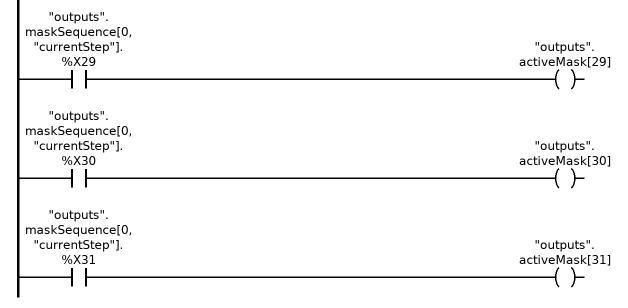
   RUNG wire#powerrail
      Contact( "outputs".maskSequence[0, "currentStep"].%X0 )
      Coil( "outputs".activeMask[0] )
   END_RUNG
   RUNG wire#powerrail
      Contact( "outputs".maskSequence[0, "currentStep"].%X1 )
      Coil( "outputs".activeMask[1] )
   END_RUNG
   RUNG wire#powerrail
      Contact( "outputs".maskSequence[0, "currentStep"].%X2 )
      Coil( "outputs".activeMask[2] )
   END_RUNG
   RUNG wire#powerrail
      Contact( "outputs".maskSequence[0, "currentStep"].%X3 )
      Coil( "outputs".activeMask[3] )
   END_RUNG
   RUNG wire#powerrail
      Contact( "outputs".maskSequence[0, "currentStep"].%X4 )
      Coil( "outputs".activeMask[4] )
   END_RUNG
   RUNG wire#powerrail
      Contact( "outputs".maskSequence[0, "currentStep"].%X5 )
      Coil( "outputs".activeMask[5] )
   END_RUNG
   RUNG wire#powerrail
      Contact( "outputs".maskSequence[0, "currentStep"].%X6 )
      Coil( "outputs".activeMask[6] )
   END_RUNG
   RUNG wire#powerrail
      Contact( "outputs".maskSequence[0, "currentStep"].%X7 )
      Coil( "outputs".activeMask[7] )
   END_RUNG
   RUNG wire#powerrail
      Contact( "outputs".maskSequence[0, "currentStep"].%X8 )
      Coil( "outputs".activeMask[8] )
   END_RUNG
   RUNG wire#powerrail
      Contact( "outputs".maskSequence[0, "currentStep"].%X9 )
      Coil( "outputs".activeMask[9] )
   END_RUNG
   RUNG wire#powerrail
      Contact( "outputs".maskSequence[0, "currentStep"].%X10 )
      Coil( "outputs".activeMask[10] )
   END_RUNG
   RUNG wire#powerrail
      Contact( "outputs".maskSequence[0, "currentStep"].%X11 )
      Coil( "outputs".activeMask[11] )
   END_RUNG
   RUNG wire#powerrail
      Contact( "outputs".maskSequence[0, "currentStep"].%X12 )
      Coil( "outputs".activeMask[12] )
   END_RUNG
   RUNG wire#powerrail
      Contact( "outputs".maskSequence[0, "currentStep"].%X13 )
      Coil( "outputs".activeMask[13] )
   END_RUNG
   RUNG wire#powerrail
      Contact( "outputs".maskSequence[0, "currentStep"].%X14 )
      Coil( "outputs".activeMask[14] )
   END_RUNG
   RUNG wire#powerrail
      Contact( "outputs".maskSequence[0, "currentStep"].%X15 )
      Coil( "outputs".activeMask[15] )
   END_RUNG
   RUNG wire#powerrail
      Contact( "outputs".maskSequence[0, "currentStep"].%X16 )
      Coil( "outputs".activeMask[16] )
   END_RUNG
   RUNG wire#powerrail
      Contact( "outputs".maskSequence[0, "currentStep"].%X17 )
      Coil( "outputs".activeMask[17] )
   END_RUNG
   RUNG wire#powerrail
      Contact( "outputs".maskSequence[0, "currentStep"].%X18 )
      Coil( "outputs".activeMask[18] )
   END_RUNG
   RUNG wire#powerrail
      Contact( "outputs".maskSequence[0, "currentStep"].%X19 )
      Coil( "outputs".activeMask[19] )
   END_RUNG
   RUNG wire#powerrail
      Contact( "outputs".maskSequence[0, "currentStep"].%X20 )
      Coil( "outputs".activeMask[20] )
   END_RUNG
   RUNG wire#powerrail
      Contact( "outputs".maskSequence[0, "currentStep"].%X21 )
      Coil( "outputs".activeMask[21] )
   END_RUNG
   RUNG wire#powerrail
      Contact( "outputs".maskSequence[0, "currentStep"].%X22 )
      Coil( "outputs".activeMask[22] )
   END_RUNG
   RUNG wire#powerrail
      Contact( "outputs".maskSequence[0, "currentStep"].%X23 )
      Coil( "outputs".activeMask[23] )
   END_RUNG
   RUNG wire#powerrail
      Contact( "outputs".maskSequence[0, "currentStep"].%X24 )
      Coil( "outputs".activeMask[24] )
   END_RUNG
   RUNG wire#powerrail
      Contact( "outputs".maskSequence[0, "currentStep"].%X25 )
      Coil( "outputs".activeMask[25] )
   END_RUNG
   RUNG wire#powerrail
      Contact( "outputs".maskSequence[0, "currentStep"].%X26 )
      Coil( "outputs".activeMask[26] )
   END_RUNG
   RUNG wire#powerrail
      Contact( "outputs".maskSequence[0, "currentStep"].%X27 )
      Coil( "outputs".activeMask[27] )
   END_RUNG
   RUNG wire#powerrail
      Contact( "outputs".maskSequence[0, "currentStep"].%X28 )
      Coil( "outputs".activeMask[28] )
   END_RUNG
   RUNG wire#powerrail
      Contact( "outputs".maskSequence[0, "currentStep"].%X29 )
      Coil( "outputs".activeMask[29] )
   END_RUNG
   RUNG wire#powerrail
      Contact( "outputs".maskSequence[0, "currentStep"].%X30 )
      Coil( "outputs".activeMask[30] )
   END_RUNG
   RUNG wire#powerrail
      Contact( "outputs".maskSequence[0, "currentStep"].%X31 )
      Coil( "outputs".activeMask[31] )
   END_RUNG
   // the same network as SCL:
   "outputs".activeMask[0] := "outputs".maskSequence[0, "currentStep"].%X0;
   "outputs".activeMask[1] := "outputs".maskSequence[0, "currentStep"].%X1;
   "outputs".activeMask[2] := "outputs".maskSequence[0, "currentStep"].%X2;
   "outputs".activeMask[3] := "outputs".maskSequence[0, "currentStep"].%X3;
   "outputs".activeMask[4] := "outputs".maskSequence[0, "currentStep"].%X4;
   "outputs".activeMask[5] := "outputs".maskSequence[0, "currentStep"].%X5;
   "outputs".activeMask[6] := "outputs".maskSequence[0, "currentStep"].%X6;
   "outputs".activeMask[7] := "outputs".maskSequence[0, "currentStep"].%X7;
   "outputs".activeMask[8] := "outputs".maskSequence[0, "currentStep"].%X8;
   "outputs".activeMask[9] := "outputs".maskSequence[0, "currentStep"].%X9;
   "outputs".activeMask[10] := "outputs".maskSequence[0, "currentStep"].%X10;
   "outputs".activeMask[11] := "outputs".maskSequence[0, "currentStep"].%X11;
   "outputs".activeMask[12] := "outputs".maskSequence[0, "currentStep"].%X12;
   "outputs".activeMask[13] := "outputs".maskSequence[0, "currentStep"].%X13;
   "outputs".activeMask[14] := "outputs".maskSequence[0, "currentStep"].%X14;
   "outputs".activeMask[15] := "outputs".maskSequence[0, "currentStep"].%X15;
   "outputs".activeMask[16] := "outputs".maskSequence[0, "currentStep"].%X16;
   "outputs".activeMask[17] := "outputs".maskSequence[0, "currentStep"].%X17;
   "outputs".activeMask[18] := "outputs".maskSequence[0, "currentStep"].%X18;
   "outputs".activeMask[19] := "outputs".maskSequence[0, "currentStep"].%X19;
   "outputs".activeMask[20] := "outputs".maskSequence[0, "currentStep"].%X20;
   "outputs".activeMask[21] := "outputs".maskSequence[0, "currentStep"].%X21;
   "outputs".activeMask[22] := "outputs".maskSequence[0, "currentStep"].%X22;
   "outputs".activeMask[23] := "outputs".maskSequence[0, "currentStep"].%X23;
   "outputs".activeMask[24] := "outputs".maskSequence[0, "currentStep"].%X24;
   "outputs".activeMask[25] := "outputs".maskSequence[0, "currentStep"].%X25;
   "outputs".activeMask[26] := "outputs".maskSequence[0, "currentStep"].%X26;
   "outputs".activeMask[27] := "outputs".maskSequence[0, "currentStep"].%X27;
   "outputs".activeMask[28] := "outputs".maskSequence[0, "currentStep"].%X28;
   "outputs".activeMask[29] := "outputs".maskSequence[0, "currentStep"].%X29;
   "outputs".activeMask[30] := "outputs".maskSequence[0, "currentStep"].%X30;
   "outputs".activeMask[31] := "outputs".maskSequence[0, "currentStep"].%X31;
END_REGION
END_FUNCTION

FUNCTION "production" : Void   // FC15, LAD
{ S7_Optimized_Access := 'TRUE' }
VERSION : 0.1
// stored: AutoNumber true, IsIECCheckEnabled false, SetENOAutomatically false, UDAEnableTagReadback false
   VAR_TEMP   // added for the SCL form of the ladder/FBD networks
      _w1 : Bool;
      _w2 : Bool;
      _w3 : Bool;
   END_VAR
BEGIN

REGION Network 1: SHIFTS PRODUCTION
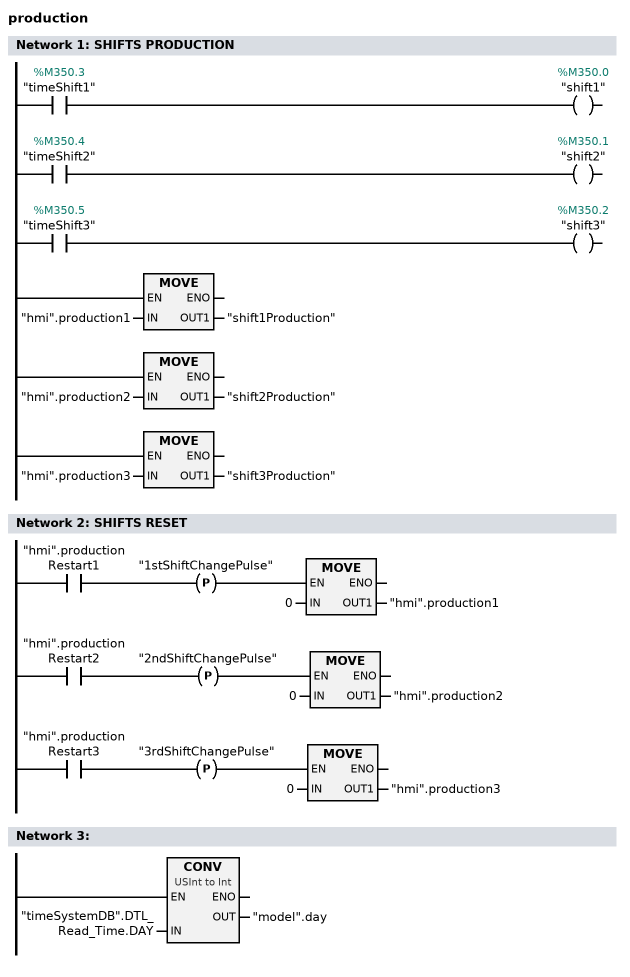
   RUNG wire#powerrail
      Contact( "timeShift1" )
      Coil( "shift1" )
   END_RUNG
   RUNG wire#powerrail
      Contact( "timeShift2" )
      Coil( "shift2" )
   END_RUNG
   RUNG wire#powerrail
      Contact( "timeShift3" )
      Coil( "shift3" )
   END_RUNG
   RUNG wire#powerrail
      Move(in := "hmi".production1, out1 => "shift1Production")
   END_RUNG
   RUNG wire#powerrail
      Move(in := "hmi".production2, out1 => "shift2Production")
   END_RUNG
   RUNG wire#powerrail
      Move(in := "hmi".production3, out1 => "shift3Production")
   END_RUNG
   // the same network as SCL:
   "shift1" := "timeShift1";
   "shift2" := "timeShift2";
   "shift3" := "timeShift3";
   "shift1Production" := "hmi".production1;
   "shift2Production" := "hmi".production2;
   "shift3Production" := "hmi".production3;
END_REGION

REGION Network 2: SHIFTS RESET
   RUNG wire#powerrail
      Contact( "hmi".productionRestart1 )
      P_Trig( "1stShiftChangePulse" )
      Move(in := 0, out1 => "hmi".production1)
   END_RUNG
   RUNG wire#powerrail
      Contact( "hmi".productionRestart2 )
      P_Trig( "2ndShiftChangePulse" )
      Move(in := 0, out1 => "hmi".production2)
   END_RUNG
   RUNG wire#powerrail
      Contact( "hmi".productionRestart3 )
      P_Trig( "3rdShiftChangePulse" )
      Move(in := 0, out1 => "hmi".production3)
   END_RUNG
   // the same network as SCL:
   #_w1 := "hmi".productionRestart1 AND NOT "1stShiftChangePulse";   // rising edge
   "1stShiftChangePulse" := "hmi".productionRestart1;
   IF #_w1 THEN "hmi".production1 := 0; END_IF;
   #_w2 := "hmi".productionRestart2 AND NOT "2ndShiftChangePulse";   // rising edge
   "2ndShiftChangePulse" := "hmi".productionRestart2;
   IF #_w2 THEN "hmi".production2 := 0; END_IF;
   #_w3 := "hmi".productionRestart3 AND NOT "3rdShiftChangePulse";   // rising edge
   "3rdShiftChangePulse" := "hmi".productionRestart3;
   IF #_w3 THEN "hmi".production3 := 0; END_IF;
END_REGION

REGION Network 3
   RUNG wire#powerrail
      { S7_Templates := "[SrcType := USInt, DestType := Int]" } Convert(in := "timeSystemDB".DTL_Read_Time.DAY, out => "model".day)
   END_RUNG
   // the same network as SCL:
   "model".day := USINT_TO_INT("timeSystemDB".DTL_Read_Time.DAY);
END_REGION
END_FUNCTION

FUNCTION "scannerConfiguration" : Void   // FC11, LAD
{ S7_Optimized_Access := 'TRUE' }
VERSION : 0.1
// stored: AutoNumber true, IsIECCheckEnabled false, SetENOAutomatically false, UDAEnableTagReadback false
   VAR_TEMP
      tempScannerOk1 : Bool;
      tempScannerOk2 : Bool;
      tempScannerOk3 : Bool;
   END_VAR
   VAR_TEMP   // added for the SCL form of the ladder/FBD networks
      _w1 : Bool;
      _w2 : Bool;
      _w3 : Bool;
      _w4 : Bool;
      _w5 : Bool;
      _w6 : Bool;
      _w7 : Bool;
      _w8 : Bool;
      _w9 : Bool;
      _w10 : Bool;
      _w11 : Bool;
      _w12 : Bool;
      _w13 : Bool;
      _w14 : Bool;
      _w15 : Bool;
   END_VAR
BEGIN

REGION Network 1: PORT CONFIGURATION
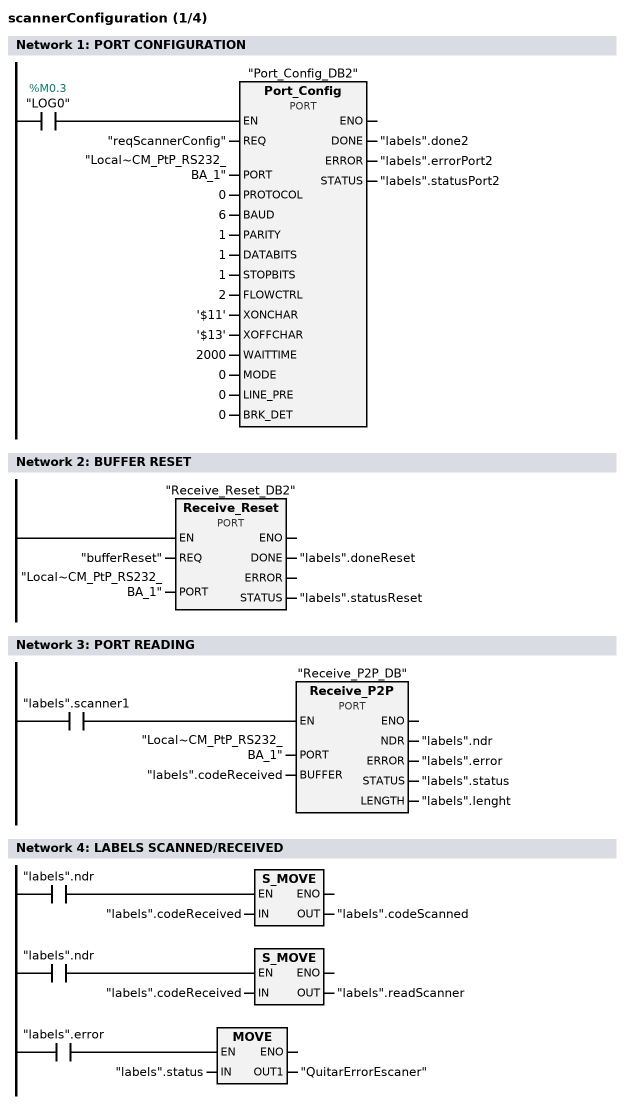
   RUNG wire#powerrail
      Contact( "LOG0" )
      { S7_Templates := "[card := 0, port_type := PORT, word_type := UInt, byte_type := USInt]" } "Port_Config_DB2".Port_Config(REQ := "reqScannerConfig", PORT := "Local~CM_PtP_RS232_BA_1", PROTOCOL := 0, BAUD := 6, PARITY := 1, DATABITS := 1, STOPBITS := 1, FLOWCTRL := 2, XONCHAR := '$11', XOFFCHAR := '$13', WAITTIME := 2000, MODE := 0, LINE_PRE := 0, BRK_DET := 0, DONE => "labels".done2, ERROR => "labels".errorPort2, STATUS => "labels".statusPort2)
   END_RUNG
   // the same network as SCL:
   IF "LOG0" THEN
       "Port_Config_DB2"(REQ := "reqScannerConfig",   // Port_Config
                         PORT := "Local~CM_PtP_RS232_BA_1",
                         PROTOCOL := 0,
                         BAUD := 6,
                         PARITY := 1,
                         DATABITS := 1,
                         STOPBITS := 1,
                         FLOWCTRL := 2,
                         XONCHAR := '$11',
                         XOFFCHAR := '$13',
                         WAITTIME := 2000,
                         MODE := 0,
                         LINE_PRE := 0,
                         BRK_DET := 0,
                         DONE => "labels".done2,
                         ERROR => "labels".errorPort2,
                         STATUS => "labels".statusPort2);
   END_IF;
END_REGION

REGION Network 2: BUFFER RESET
   RUNG wire#powerrail
      { S7_Templates := "[card := 0, port_type := PORT]" } "Receive_Reset_DB2".Receive_Reset(REQ := "bufferReset", PORT := "Local~CM_PtP_RS232_BA_1", DONE => "labels".doneReset, ERROR =>, STATUS => "labels".statusReset)
   END_RUNG
   // the same network as SCL:
   "Receive_Reset_DB2"(REQ := "bufferReset",   // Receive_Reset
                       PORT := "Local~CM_PtP_RS232_BA_1",
                       DONE => "labels".doneReset,
                       STATUS => "labels".statusReset);
END_REGION

REGION Network 3: PORT READING
   RUNG wire#powerrail
      Contact( "labels".scanner1 )
      { S7_Templates := "[card := 0, port_type := PORT, word_type := UInt, any_type := Variant]" } "Receive_P2P_DB".Receive_P2P(PORT := "Local~CM_PtP_RS232_BA_1", BUFFER := "labels".codeReceived, NDR => "labels".ndr, ERROR => "labels".error, STATUS => "labels".status, LENGTH => "labels".lenght)
   END_RUNG
   // the same network as SCL:
   IF "labels".scanner1 THEN
       "Receive_P2P_DB"(PORT := "Local~CM_PtP_RS232_BA_1",   // Receive_P2P
                        BUFFER := "labels".codeReceived,
                        NDR => "labels".ndr,
                        ERROR => "labels".error,
                        STATUS => "labels".status,
                        LENGTH => "labels".lenght);
   END_IF;
END_REGION

REGION Network 4: LABELS SCANNED/RECEIVED
   RUNG wire#powerrail
      Contact( "labels".ndr )
      S_Move(in := "labels".codeReceived, out => "labels".codeScanned)
   END_RUNG
   RUNG wire#powerrail
      Contact( "labels".ndr )
      S_Move(in := "labels".codeReceived, out => "labels".readScanner)
   END_RUNG
   RUNG wire#powerrail
      Contact( "labels".error )
      Move(in := "labels".status, out1 => "QuitarErrorEscaner")
   END_RUNG
   // the same network as SCL:
   IF "labels".ndr THEN
       "labels".codeScanned := "labels".codeReceived;
       "labels".readScanner := "labels".codeReceived;
   END_IF;
   IF "labels".error THEN "QuitarErrorEscaner" := "labels".status; END_IF;
END_REGION

REGION Network 5: SCANNER COMPARISON
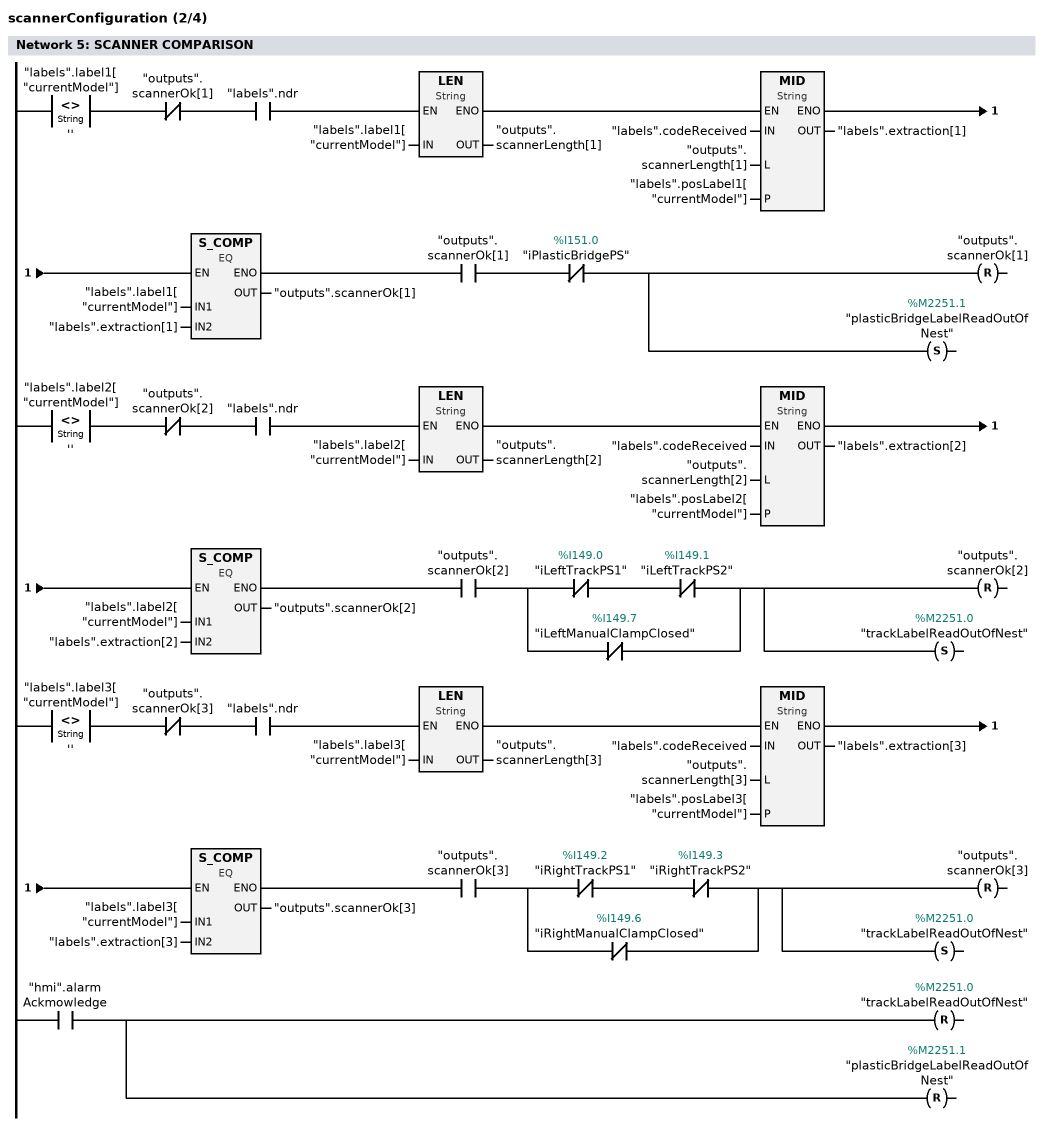
   RUNG wire#powerrail
      { S7_Templates := "SrcType := String" } NE_Contact(in1 := "labels".label1["currentModel"], in2 := '')
      I_Contact( "outputs".scannerOk[1] )
      Contact( "labels".ndr )
      { S7_Templates := "[str_type := String, return_type := Int]" } LEN(IN := "labels".label1["currentModel"], OUT => "outputs".scannerLength[1])
      { S7_Templates := "value_type := String" } MID(IN := "labels".codeReceived, L := "outputs".scannerLength[1], P := "labels".posLabel1["currentModel"], OUT => "labels".extraction[1])
      { S7_Templates := "[relation := EQ, src_type := String]" } S_COMP(IN1 := "labels".label1["currentModel"], IN2 := "labels".extraction[1], OUT => "outputs".scannerOk[1])
      Contact( "outputs".scannerOk[1] )
      I_Contact( "iPlasticBridgePS" )
      wire#w1
      R_Coil( "outputs".scannerOk[1] )
   END_RUNG
   RUNG wire#w1
      S_Coil( "plasticBridgeLabelReadOutOfNest" )
   END_RUNG
   RUNG wire#powerrail
      { S7_Templates := "SrcType := String" } NE_Contact(in1 := "labels".label2["currentModel"], in2 := '')
      I_Contact( "outputs".scannerOk[2] )
      Contact( "labels".ndr )
      { S7_Templates := "[str_type := String, return_type := Int]" } LEN(IN := "labels".label2["currentModel"], OUT => "outputs".scannerLength[2])
      { S7_Templates := "value_type := String" } MID(IN := "labels".codeReceived, L := "outputs".scannerLength[2], P := "labels".posLabel2["currentModel"], OUT => "labels".extraction[2])
      { S7_Templates := "[relation := EQ, src_type := String]" } S_COMP(IN1 := "labels".label2["currentModel"], IN2 := "labels".extraction[2], OUT => "outputs".scannerOk[2])
      Contact( "outputs".scannerOk[2] )
      wire#w2
      I_Contact( "iLeftTrackPS1" )
      I_Contact( "iLeftTrackPS2" )
      wire#w3
      R_Coil( "outputs".scannerOk[2] )
   END_RUNG
   RUNG wire#w2
      I_Contact( "iLeftManualClampClosed" )
   END_RUNG wire#w3
   RUNG wire#w3
      S_Coil( "trackLabelReadOutOfNest" )
   END_RUNG
   RUNG wire#powerrail
      { S7_Templates := "SrcType := String" } NE_Contact(in1 := "labels".label3["currentModel"], in2 := '')
      I_Contact( "outputs".scannerOk[3] )
      Contact( "labels".ndr )
      { S7_Templates := "[str_type := String, return_type := Int]" } LEN(IN := "labels".label3["currentModel"], OUT => "outputs".scannerLength[3])
      { S7_Templates := "value_type := String" } MID(IN := "labels".codeReceived, L := "outputs".scannerLength[3], P := "labels".posLabel3["currentModel"], OUT => "labels".extraction[3])
      { S7_Templates := "[relation := EQ, src_type := String]" } S_COMP(IN1 := "labels".label3["currentModel"], IN2 := "labels".extraction[3], OUT => "outputs".scannerOk[3])
      Contact( "outputs".scannerOk[3] )
      wire#w4
      I_Contact( "iRightTrackPS1" )
      I_Contact( "iRightTrackPS2" )
      wire#w5
      R_Coil( "outputs".scannerOk[3] )
   END_RUNG
   RUNG wire#w4
      I_Contact( "iRightManualClampClosed" )
   END_RUNG wire#w5
   RUNG wire#w5
      S_Coil( "trackLabelReadOutOfNest" )
   END_RUNG
   RUNG wire#powerrail
      Contact( "hmi".alarmAckmowledge )
      wire#w6
      R_Coil( "trackLabelReadOutOfNest" )
   END_RUNG
   RUNG wire#w6
      R_Coil( "plasticBridgeLabelReadOutOfNest" )
   END_RUNG
   // the same network as SCL:
   #_w1 := ("labels".label1["currentModel"] <> '') AND NOT "outputs".scannerOk[1] AND "labels".ndr;
   LEN(EN := #_w1, IN := "labels".label1["currentModel"], OUT => "outputs".scannerLength[1], ENO => #_w2);
   MID(EN := #_w2,
       IN := "labels".codeReceived,
       L := "outputs".scannerLength[1],
       P := "labels".posLabel1["currentModel"],
       OUT => "labels".extraction[1],
       ENO => #_w3);
   S_COMP(EN := #_w3,
          IN1 := "labels".label1["currentModel"],
          IN2 := "labels".extraction[1],
          OUT => "outputs".scannerOk[1],
          ENO => #_w4);
   #_w5 := #_w4 AND "outputs".scannerOk[1] AND NOT "iPlasticBridgePS";
   IF #_w5 THEN
       "outputs".scannerOk[1] := FALSE;
       "plasticBridgeLabelReadOutOfNest" := TRUE;
   END_IF;
   #_w6 := ("labels".label2["currentModel"] <> '') AND NOT "outputs".scannerOk[2] AND "labels".ndr;
   LEN(EN := #_w6, IN := "labels".label2["currentModel"], OUT => "outputs".scannerLength[2], ENO => #_w7);
   MID(EN := #_w7,
       IN := "labels".codeReceived,
       L := "outputs".scannerLength[2],
       P := "labels".posLabel2["currentModel"],
       OUT => "labels".extraction[2],
       ENO => #_w8);
   S_COMP(EN := #_w8,
          IN1 := "labels".label2["currentModel"],
          IN2 := "labels".extraction[2],
          OUT => "outputs".scannerOk[2],
          ENO => #_w9);
   #_w10 := #_w9 AND "outputs".scannerOk[2] AND ((NOT "iLeftTrackPS1" AND NOT "iLeftTrackPS2") OR NOT "iLeftManualClampClosed");
   IF #_w10 THEN
       "outputs".scannerOk[2] := FALSE;
       "trackLabelReadOutOfNest" := TRUE;
   END_IF;
   #_w11 := ("labels".label3["currentModel"] <> '') AND NOT "outputs".scannerOk[3] AND "labels".ndr;
   LEN(EN := #_w11, IN := "labels".label3["currentModel"], OUT => "outputs".scannerLength[3], ENO => #_w12);
   MID(EN := #_w12,
       IN := "labels".codeReceived,
       L := "outputs".scannerLength[3],
       P := "labels".posLabel3["currentModel"],
       OUT => "labels".extraction[3],
       ENO => #_w13);
   S_COMP(EN := #_w13,
          IN1 := "labels".label3["currentModel"],
          IN2 := "labels".extraction[3],
          OUT => "outputs".scannerOk[3],
          ENO => #_w14);
   #_w15 := #_w14 AND "outputs".scannerOk[3] AND ((NOT "iRightTrackPS1" AND NOT "iRightTrackPS2") OR NOT "iRightManualClampClosed");
   IF #_w15 THEN
       "outputs".scannerOk[3] := FALSE;
       "trackLabelReadOutOfNest" := TRUE;
   END_IF;
   IF "hmi".alarmAckmowledge THEN
       "trackLabelReadOutOfNest" := FALSE;
       "plasticBridgeLabelReadOutOfNest" := FALSE;
   END_IF;
END_REGION

REGION Network 6: CHANGE OF STEP SCANNER RESET
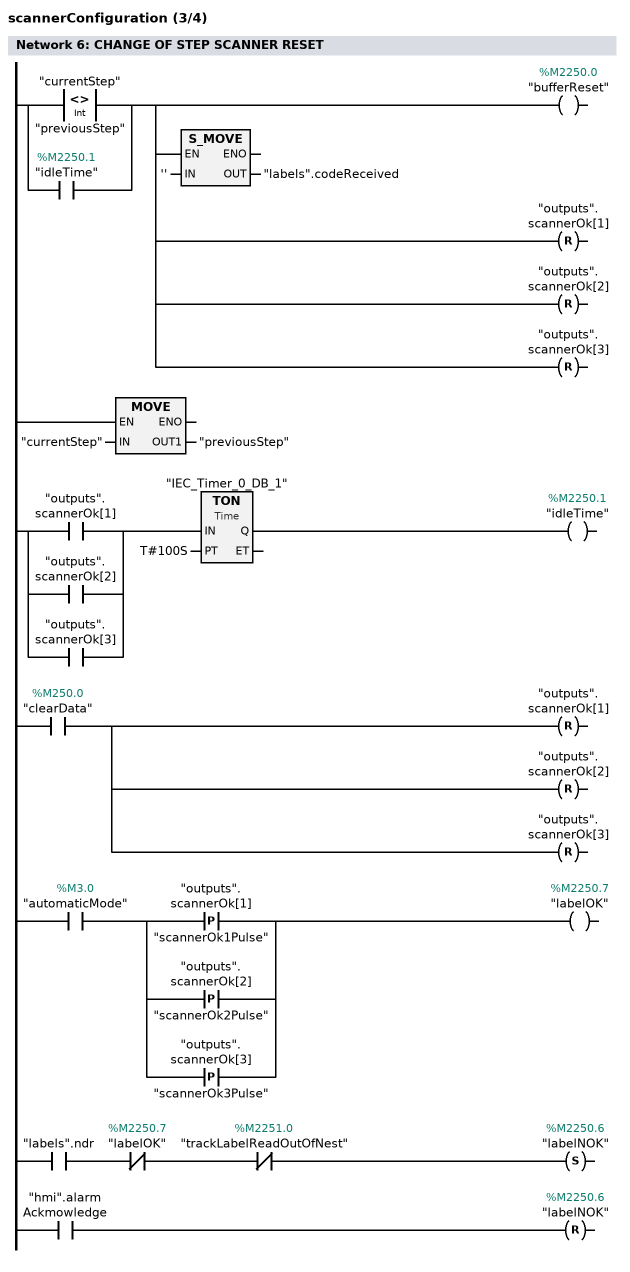
   RUNG wire#powerrail
      { S7_Templates := "SrcType := Int" } NE_Contact(in1 := "currentStep", in2 := "previousStep")
      wire#w1
      Coil( "bufferReset" )
   END_RUNG
   RUNG wire#powerrail
      Contact( "idleTime" )
   END_RUNG wire#w1
   RUNG wire#w1
      S_Move(in := '', out => "labels".codeReceived)
   END_RUNG
   RUNG wire#w1
      R_Coil( "outputs".scannerOk[1] )
   END_RUNG
   RUNG wire#w1
      R_Coil( "outputs".scannerOk[2] )
   END_RUNG
   RUNG wire#w1
      R_Coil( "outputs".scannerOk[3] )
   END_RUNG
   RUNG wire#powerrail
      Move(in := "currentStep", out1 => "previousStep")
   END_RUNG
   RUNG wire#powerrail
      Contact( "outputs".scannerOk[1] )
      wire#w2
      { S7_Templates := "time_type := Time" } "IEC_Timer_0_DB_1".TON(pt := T#100S, et =>)
      Coil( "idleTime" )
   END_RUNG
   RUNG wire#powerrail
      Contact( "outputs".scannerOk[2] )
   END_RUNG wire#w2
   RUNG wire#powerrail
      Contact( "outputs".scannerOk[3] )
   END_RUNG wire#w2
   RUNG wire#powerrail
      Contact( "clearData" )
      wire#w3
      R_Coil( "outputs".scannerOk[1] )
   END_RUNG
   RUNG wire#w3
      R_Coil( "outputs".scannerOk[2] )
   END_RUNG
   RUNG wire#w3
      R_Coil( "outputs".scannerOk[3] )
   END_RUNG
   RUNG wire#powerrail
      Contact( "automaticMode" )
      wire#w4
      P_Contact(operand := "outputs".scannerOk[1], bit := "scannerOk1Pulse")
      wire#w5
      Coil( "labelOK" )
   END_RUNG
   RUNG wire#w4
      P_Contact(operand := "outputs".scannerOk[2], bit := "scannerOk2Pulse")
   END_RUNG wire#w5
   RUNG wire#w4
      P_Contact(operand := "outputs".scannerOk[3], bit := "scannerOk3Pulse")
   END_RUNG wire#w5
   RUNG wire#powerrail
      Contact( "labels".ndr )
      I_Contact( "labelOK" )
      I_Contact( "trackLabelReadOutOfNest" )
      S_Coil( "labelNOK" )
   END_RUNG
   RUNG wire#powerrail
      Contact( "hmi".alarmAckmowledge )
      R_Coil( "labelNOK" )
   END_RUNG
   // the same network as SCL:
   "bufferReset" := ("currentStep" <> "previousStep") OR "idleTime";
   IF "bufferReset" THEN
       "labels".codeReceived := '';
       "outputs".scannerOk[1] := FALSE;
       "outputs".scannerOk[2] := FALSE;
       "outputs".scannerOk[3] := FALSE;
   END_IF;
   "previousStep" := "currentStep";
   "IEC_Timer_0_DB_1".TON(IN := "outputs".scannerOk[1] OR "outputs".scannerOk[2] OR "outputs".scannerOk[3],
                          PT := T#100S);
   "idleTime" := "IEC_Timer_0_DB_1".Q;
   IF "clearData" THEN
       "outputs".scannerOk[1] := FALSE;
       "outputs".scannerOk[2] := FALSE;
       "outputs".scannerOk[3] := FALSE;
   END_IF;
   #_w1 := "automaticMode" AND "outputs".scannerOk[1] AND NOT "scannerOk1Pulse";   // rising edge of "outputs".scannerOk[1]
   "scannerOk1Pulse" := "outputs".scannerOk[1];
   #_w2 := "automaticMode" AND "outputs".scannerOk[2] AND NOT "scannerOk2Pulse";   // rising edge of "outputs".scannerOk[2]
   "scannerOk2Pulse" := "outputs".scannerOk[2];
   #_w3 := "automaticMode" AND "outputs".scannerOk[3] AND NOT "scannerOk3Pulse";   // rising edge of "outputs".scannerOk[3]
   "scannerOk3Pulse" := "outputs".scannerOk[3];
   "labelOK" := #_w1 OR #_w2 OR #_w3;
   IF "labels".ndr AND NOT "labelOK" AND NOT "trackLabelReadOutOfNest" THEN "labelNOK" := TRUE; END_IF;
   IF "hmi".alarmAckmowledge THEN "labelNOK" := FALSE; END_IF;
END_REGION

REGION Network 7: SCANNER DATA LOG
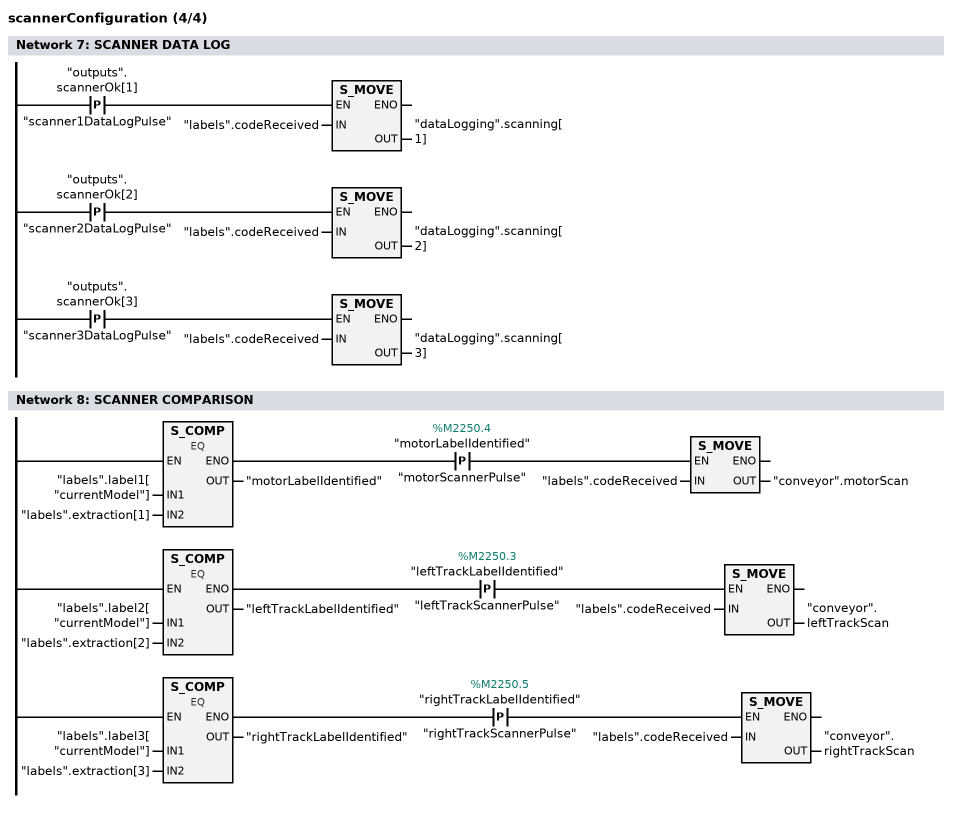
   RUNG wire#powerrail
      P_Contact(operand := "outputs".scannerOk[1], bit := "scanner1DataLogPulse")
      S_Move(in := "labels".codeReceived, out => "dataLogging".scanning[1])
   END_RUNG
   RUNG wire#powerrail
      P_Contact(operand := "outputs".scannerOk[2], bit := "scanner2DataLogPulse")
      S_Move(in := "labels".codeReceived, out => "dataLogging".scanning[2])
   END_RUNG
   RUNG wire#powerrail
      P_Contact(operand := "outputs".scannerOk[3], bit := "scanner3DataLogPulse")
      S_Move(in := "labels".codeReceived, out => "dataLogging".scanning[3])
   END_RUNG
   // the same network as SCL:
   #_w1 := "outputs".scannerOk[1] AND NOT "scanner1DataLogPulse";   // rising edge of "outputs".scannerOk[1]
   "scanner1DataLogPulse" := "outputs".scannerOk[1];
   IF #_w1 THEN "dataLogging".scanning[1] := "labels".codeReceived; END_IF;
   #_w2 := "outputs".scannerOk[2] AND NOT "scanner2DataLogPulse";   // rising edge of "outputs".scannerOk[2]
   "scanner2DataLogPulse" := "outputs".scannerOk[2];
   IF #_w2 THEN "dataLogging".scanning[2] := "labels".codeReceived; END_IF;
   #_w3 := "outputs".scannerOk[3] AND NOT "scanner3DataLogPulse";   // rising edge of "outputs".scannerOk[3]
   "scanner3DataLogPulse" := "outputs".scannerOk[3];
   IF #_w3 THEN "dataLogging".scanning[3] := "labels".codeReceived; END_IF;
END_REGION

REGION Network 8: SCANNER COMPARISON
   RUNG wire#powerrail
      { S7_Templates := "[relation := EQ, src_type := String]" } S_COMP(IN1 := "labels".label1["currentModel"], IN2 := "labels".extraction[1], OUT => "motorLabelIdentified")
      P_Contact(operand := "motorLabelIdentified", bit := "motorScannerPulse")
      S_Move(in := "labels".codeReceived, out => "conveyor".motorScan)
   END_RUNG
   RUNG wire#powerrail
      { S7_Templates := "[relation := EQ, src_type := String]" } S_COMP(IN1 := "labels".label2["currentModel"], IN2 := "labels".extraction[2], OUT => "leftTrackLabelIdentified")
      P_Contact(operand := "leftTrackLabelIdentified", bit := "leftTrackScannerPulse")
      S_Move(in := "labels".codeReceived, out => "conveyor".leftTrackScan)
   END_RUNG
   RUNG wire#powerrail
      { S7_Templates := "[relation := EQ, src_type := String]" } S_COMP(IN1 := "labels".label3["currentModel"], IN2 := "labels".extraction[3], OUT => "rightTrackLabelIdentified")
      P_Contact(operand := "rightTrackLabelIdentified", bit := "rightTrackScannerPulse")
      S_Move(in := "labels".codeReceived, out => "conveyor".rightTrackScan)
   END_RUNG
   // the same network as SCL:
   S_COMP(IN1 := "labels".label1["currentModel"],
          IN2 := "labels".extraction[1],
          OUT => "motorLabelIdentified",
          ENO => #_w1);
   #_w2 := #_w1 AND "motorLabelIdentified" AND NOT "motorScannerPulse";   // rising edge of "motorLabelIdentified"
   "motorScannerPulse" := "motorLabelIdentified";
   IF #_w2 THEN "conveyor".motorScan := "labels".codeReceived; END_IF;
   S_COMP(IN1 := "labels".label2["currentModel"],
          IN2 := "labels".extraction[2],
          OUT => "leftTrackLabelIdentified",
          ENO => #_w3);
   #_w4 := #_w3 AND "leftTrackLabelIdentified" AND NOT "leftTrackScannerPulse";   // rising edge of "leftTrackLabelIdentified"
   "leftTrackScannerPulse" := "leftTrackLabelIdentified";
   IF #_w4 THEN "conveyor".leftTrackScan := "labels".codeReceived; END_IF;
   S_COMP(IN1 := "labels".label3["currentModel"],
          IN2 := "labels".extraction[3],
          OUT => "rightTrackLabelIdentified",
          ENO => #_w5);
   #_w6 := #_w5 AND "rightTrackLabelIdentified" AND NOT "rightTrackScannerPulse";   // rising edge of "rightTrackLabelIdentified"
   "rightTrackScannerPulse" := "rightTrackLabelIdentified";
   IF #_w6 THEN "conveyor".rightTrackScan := "labels".codeReceived; END_IF;
END_REGION
END_FUNCTION

FUNCTION "stationAlarms" : Void   // FC2, LAD
{ S7_Optimized_Access := 'TRUE' }
VERSION : 0.1
// stored: AutoNumber true, IsIECCheckEnabled false, SetENOAutomatically false, UDAEnableTagReadback false
   VAR_TEMP
      visualizationDefault : Bool;
   END_VAR
   VAR_TEMP   // added for the SCL form of the ladder/FBD networks
      _w1 : Bool;
      _w2 : Bool;
      _w3 : Bool;
      _w4 : Bool;
      _w5 : Bool;
   END_VAR
BEGIN

REGION Network 1: Visualization Defaults
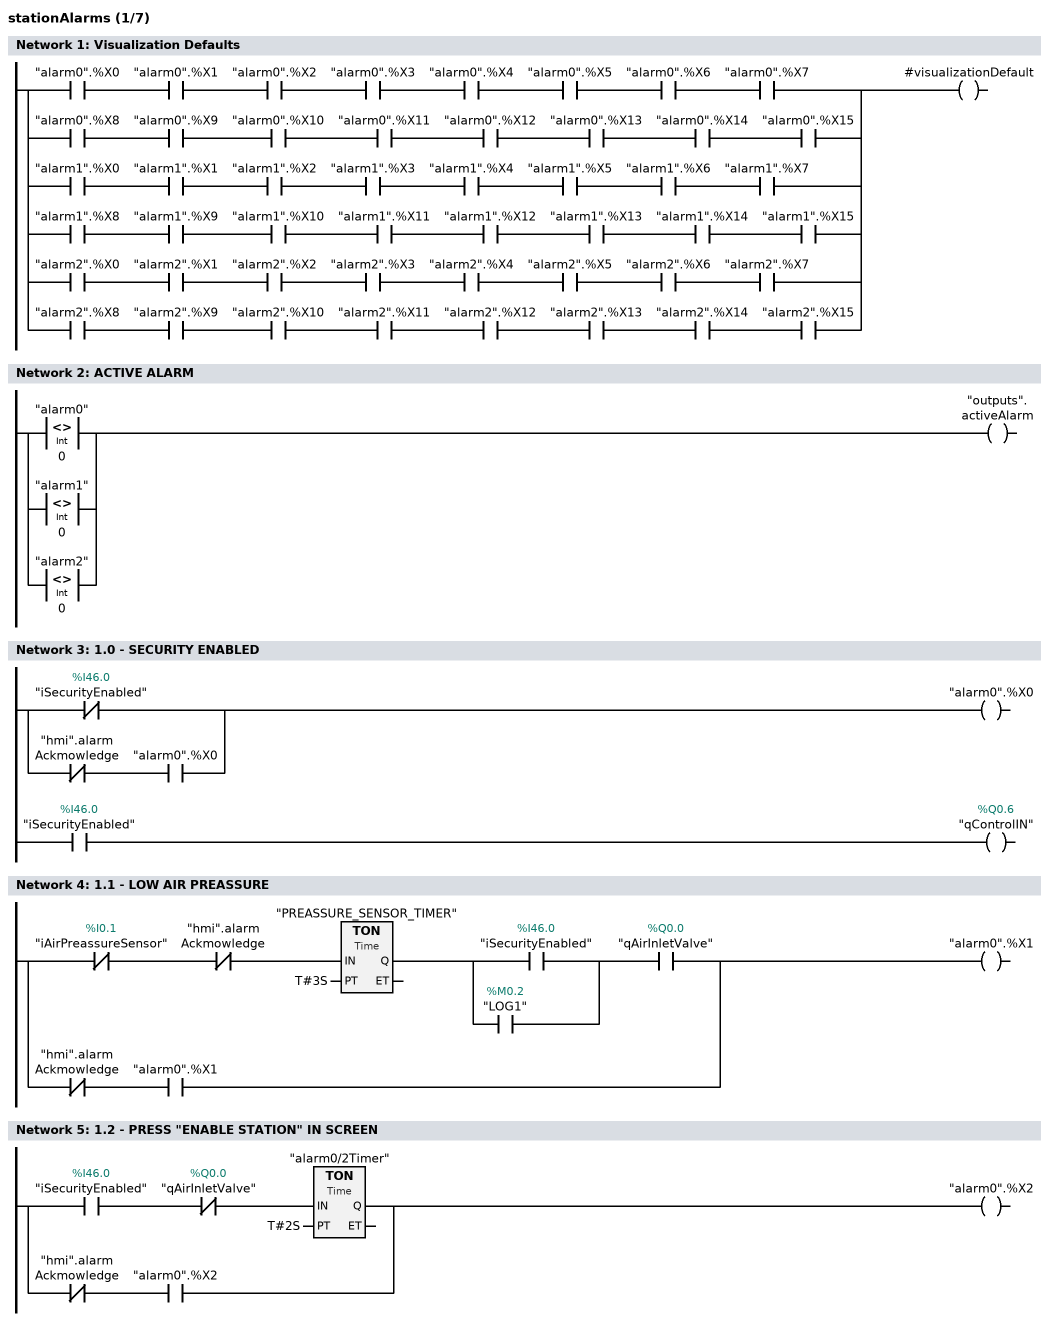
   RUNG wire#powerrail
      Contact( "alarm0".%X0 )
      Contact( "alarm0".%X1 )
      Contact( "alarm0".%X2 )
      Contact( "alarm0".%X3 )
      Contact( "alarm0".%X4 )
      Contact( "alarm0".%X5 )
      Contact( "alarm0".%X6 )
      Contact( "alarm0".%X7 )
      wire#w1
      Coil( #visualizationDefault )
   END_RUNG
   RUNG wire#powerrail
      Contact( "alarm0".%X8 )
      Contact( "alarm0".%X9 )
      Contact( "alarm0".%X10 )
      Contact( "alarm0".%X11 )
      Contact( "alarm0".%X12 )
      Contact( "alarm0".%X13 )
      Contact( "alarm0".%X14 )
      Contact( "alarm0".%X15 )
   END_RUNG wire#w1
   RUNG wire#powerrail
      Contact( "alarm1".%X0 )
      Contact( "alarm1".%X1 )
      Contact( "alarm1".%X2 )
      Contact( "alarm1".%X3 )
      Contact( "alarm1".%X4 )
      Contact( "alarm1".%X5 )
      Contact( "alarm1".%X6 )
      Contact( "alarm1".%X7 )
   END_RUNG wire#w1
   RUNG wire#powerrail
      Contact( "alarm1".%X8 )
      Contact( "alarm1".%X9 )
      Contact( "alarm1".%X10 )
      Contact( "alarm1".%X11 )
      Contact( "alarm1".%X12 )
      Contact( "alarm1".%X13 )
      Contact( "alarm1".%X14 )
      Contact( "alarm1".%X15 )
   END_RUNG wire#w1
   RUNG wire#powerrail
      Contact( "alarm2".%X0 )
      Contact( "alarm2".%X1 )
      Contact( "alarm2".%X2 )
      Contact( "alarm2".%X3 )
      Contact( "alarm2".%X4 )
      Contact( "alarm2".%X5 )
      Contact( "alarm2".%X6 )
      Contact( "alarm2".%X7 )
   END_RUNG wire#w1
   RUNG wire#powerrail
      Contact( "alarm2".%X8 )
      Contact( "alarm2".%X9 )
      Contact( "alarm2".%X10 )
      Contact( "alarm2".%X11 )
      Contact( "alarm2".%X12 )
      Contact( "alarm2".%X13 )
      Contact( "alarm2".%X14 )
      Contact( "alarm2".%X15 )
   END_RUNG wire#w1
   // the same network as SCL:
   #visualizationDefault := ("alarm0".%X0 AND "alarm0".%X1 AND "alarm0".%X2 AND "alarm0".%X3 AND "alarm0".%X4 AND "alarm0".%X5 AND "alarm0".%X6 AND "alarm0".%X7) OR ("alarm0".%X8 AND "alarm0".%X9 AND "alarm0".%X10 AND "alarm0".%X11 AND "alarm0".%X12 AND "alarm0".%X13 AND "alarm0".%X14 AND "alarm0".%X15) OR ("alarm1".%X0 AND "alarm1".%X1 AND "alarm1".%X2 AND "alarm1".%X3 AND "alarm1".%X4 AND "alarm1".%X5 AND "alarm1".%X6 AND "alarm1".%X7) OR ("alarm1".%X8 AND "alarm1".%X9 AND "alarm1".%X10 AND "alarm1".%X11 AND "alarm1".%X12 AND "alarm1".%X13 AND "alarm1".%X14 AND "alarm1".%X15) OR ("alarm2".%X0 AND "alarm2".%X1 AND "alarm2".%X2 AND "alarm2".%X3 AND "alarm2".%X4 AND "alarm2".%X5 AND "alarm2".%X6 AND "alarm2".%X7) OR ("alarm2".%X8 AND "alarm2".%X9 AND "alarm2".%X10 AND "alarm2".%X11 AND "alarm2".%X12 AND "alarm2".%X13 AND "alarm2".%X14 AND "alarm2".%X15);
END_REGION

REGION Network 2: ACTIVE ALARM
   RUNG wire#powerrail
      { S7_Templates := "SrcType := Int" } NE_Contact(in1 := "alarm0", in2 := 0)
      wire#w1
      Coil( "outputs".activeAlarm )
   END_RUNG
   RUNG wire#powerrail
      { S7_Templates := "SrcType := Int" } NE_Contact(in1 := "alarm1", in2 := 0)
   END_RUNG wire#w1
   RUNG wire#powerrail
      { S7_Templates := "SrcType := Int" } NE_Contact(in1 := "alarm2", in2 := 0)
   END_RUNG wire#w1
   // the same network as SCL:
   "outputs".activeAlarm := ("alarm0" <> 0) OR ("alarm1" <> 0) OR ("alarm2" <> 0);
END_REGION

REGION Network 3: 1.0 - SECURITY ENABLED
   RUNG wire#powerrail
      I_Contact( "iSecurityEnabled" )
      wire#w1
      Coil( "alarm0".%X0 )
   END_RUNG
   RUNG wire#powerrail
      I_Contact( "hmi".alarmAckmowledge )
      Contact( "alarm0".%X0 )
   END_RUNG wire#w1
   RUNG wire#powerrail
      Contact( "iSecurityEnabled" )
      Coil( "qControlIN" )
   END_RUNG
   // the same network as SCL:
   "alarm0".%X0 := NOT "iSecurityEnabled" OR (NOT "hmi".alarmAckmowledge AND "alarm0".%X0);
   "qControlIN" := "iSecurityEnabled";
END_REGION

REGION Network 4: 1.1 - LOW AIR PREASSURE
   RUNG wire#powerrail
      I_Contact( "iAirPreassureSensor" )
      I_Contact( "hmi".alarmAckmowledge )
      { S7_Templates := "time_type := Time" } "PREASSURE_SENSOR_TIMER".TON(pt := T#3S, et =>)
      wire#w1
      Contact( "iSecurityEnabled" )
      wire#w2
      Contact( "qAirInletValve" )
      wire#w3
      Coil( "alarm0".%X1 )
   END_RUNG
   RUNG wire#w1
      Contact( "LOG1" )
   END_RUNG wire#w2
   RUNG wire#powerrail
      I_Contact( "hmi".alarmAckmowledge )
      Contact( "alarm0".%X1 )
   END_RUNG wire#w3
   // the same network as SCL:
   "PREASSURE_SENSOR_TIMER".TON(IN := NOT "iAirPreassureSensor" AND NOT "hmi".alarmAckmowledge, PT := T#3S);
   "alarm0".%X1 := ("PREASSURE_SENSOR_TIMER".Q AND ("iSecurityEnabled" OR "LOG1") AND "qAirInletValve") OR (NOT "hmi".alarmAckmowledge AND "alarm0".%X1);
END_REGION

REGION Network 5: 1.2 - PRESS "ENABLE STATION" IN SCREEN
   RUNG wire#powerrail
      Contact( "iSecurityEnabled" )
      I_Contact( "qAirInletValve" )
      { S7_Templates := "time_type := Time" } "alarm0/2Timer".TON(pt := T#2S, et =>)
      wire#w1
      Coil( "alarm0".%X2 )
   END_RUNG
   RUNG wire#powerrail
      I_Contact( "hmi".alarmAckmowledge )
      Contact( "alarm0".%X2 )
   END_RUNG wire#w1
   // the same network as SCL:
   "alarm0/2Timer".TON(IN := "iSecurityEnabled" AND NOT "qAirInletValve", PT := T#2S);
   "alarm0".%X2 := "alarm0/2Timer".Q OR (NOT "hmi".alarmAckmowledge AND "alarm0".%X2);
END_REGION

REGION Network 6: 1.3 - ESTOP PRESSED
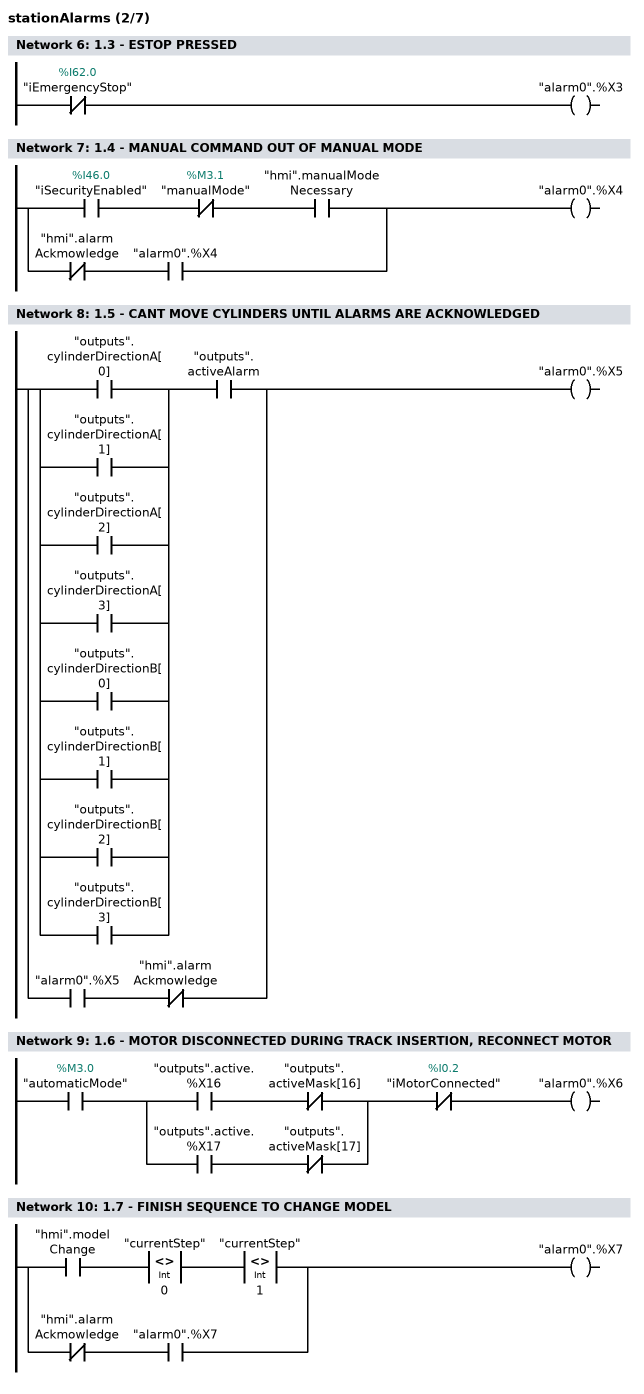
   RUNG wire#powerrail
      I_Contact( "iEmergencyStop" )
      Coil( "alarm0".%X3 )
   END_RUNG
   // the same network as SCL:
   "alarm0".%X3 := NOT "iEmergencyStop";
END_REGION

REGION Network 7: 1.4 - MANUAL COMMAND OUT OF MANUAL MODE
   RUNG wire#powerrail
      Contact( "iSecurityEnabled" )
      I_Contact( "manualMode" )
      Contact( "hmi".manualModeNecessary )
      wire#w1
      Coil( "alarm0".%X4 )
   END_RUNG
   RUNG wire#powerrail
      I_Contact( "hmi".alarmAckmowledge )
      Contact( "alarm0".%X4 )
   END_RUNG wire#w1
   // the same network as SCL:
   "alarm0".%X4 := ("iSecurityEnabled" AND NOT "manualMode" AND "hmi".manualModeNecessary) OR (NOT "hmi".alarmAckmowledge AND "alarm0".%X4);
END_REGION

REGION Network 8: 1.5 - CANT MOVE CYLINDERS UNTIL ALARMS ARE ACKNOWLEDGED
   RUNG wire#powerrail
      Contact( "outputs".cylinderDirectionA[0] )
      wire#w1
      Contact( "outputs".activeAlarm )
      wire#w2
      Coil( "alarm0".%X5 )
   END_RUNG
   RUNG wire#powerrail
      Contact( "outputs".cylinderDirectionA[1] )
   END_RUNG wire#w1
   RUNG wire#powerrail
      Contact( "outputs".cylinderDirectionA[2] )
   END_RUNG wire#w1
   RUNG wire#powerrail
      Contact( "outputs".cylinderDirectionA[3] )
   END_RUNG wire#w1
   RUNG wire#powerrail
      Contact( "outputs".cylinderDirectionB[0] )
   END_RUNG wire#w1
   RUNG wire#powerrail
      Contact( "outputs".cylinderDirectionB[1] )
   END_RUNG wire#w1
   RUNG wire#powerrail
      Contact( "outputs".cylinderDirectionB[2] )
   END_RUNG wire#w1
   RUNG wire#powerrail
      Contact( "outputs".cylinderDirectionB[3] )
   END_RUNG wire#w1
   RUNG wire#powerrail
      Contact( "alarm0".%X5 )
      I_Contact( "hmi".alarmAckmowledge )
   END_RUNG wire#w2
   // the same network as SCL:
   "alarm0".%X5 := (("outputs".cylinderDirectionA[0] OR "outputs".cylinderDirectionA[1] OR "outputs".cylinderDirectionA[2] OR "outputs".cylinderDirectionA[3] OR "outputs".cylinderDirectionB[0] OR "outputs".cylinderDirectionB[1] OR "outputs".cylinderDirectionB[2] OR "outputs".cylinderDirectionB[3]) AND "outputs".activeAlarm) OR ("alarm0".%X5 AND NOT "hmi".alarmAckmowledge);
END_REGION

REGION Network 9: 1.6 - MOTOR DISCONNECTED DURING TRACK INSERTION, RECONNECT MOTOR
   RUNG wire#powerrail
      Contact( "automaticMode" )
      wire#w1
      Contact( "outputs".active.%X16 )
      I_Contact( "outputs".activeMask[16] )
      wire#w2
      I_Contact( "iMotorConnected" )
      Coil( "alarm0".%X6 )
   END_RUNG
   RUNG wire#w1
      Contact( "outputs".active.%X17 )
      I_Contact( "outputs".activeMask[17] )
   END_RUNG wire#w2
   // the same network as SCL:
   "alarm0".%X6 := "automaticMode" AND (("outputs".active.%X16 AND NOT "outputs".activeMask[16]) OR ("outputs".active.%X17 AND NOT "outputs".activeMask[17])) AND NOT "iMotorConnected";
END_REGION

REGION Network 10: 1.7 - FINISH SEQUENCE TO CHANGE MODEL
   RUNG wire#powerrail
      Contact( "hmi".modelChange )
      { S7_Templates := "SrcType := Int" } NE_Contact(in1 := "currentStep", in2 := 0)
      { S7_Templates := "SrcType := Int" } NE_Contact(in1 := "currentStep", in2 := 1)
      wire#w1
      Coil( "alarm0".%X7 )
   END_RUNG
   RUNG wire#powerrail
      I_Contact( "hmi".alarmAckmowledge )
      Contact( "alarm0".%X7 )
   END_RUNG wire#w1
   // the same network as SCL:
   "alarm0".%X7 := ("hmi".modelChange AND ("currentStep" <> 0) AND ("currentStep" <> 1)) OR (NOT "hmi".alarmAckmowledge AND "alarm0".%X7);
END_REGION

REGION Network 11: 1.8 - SPARE
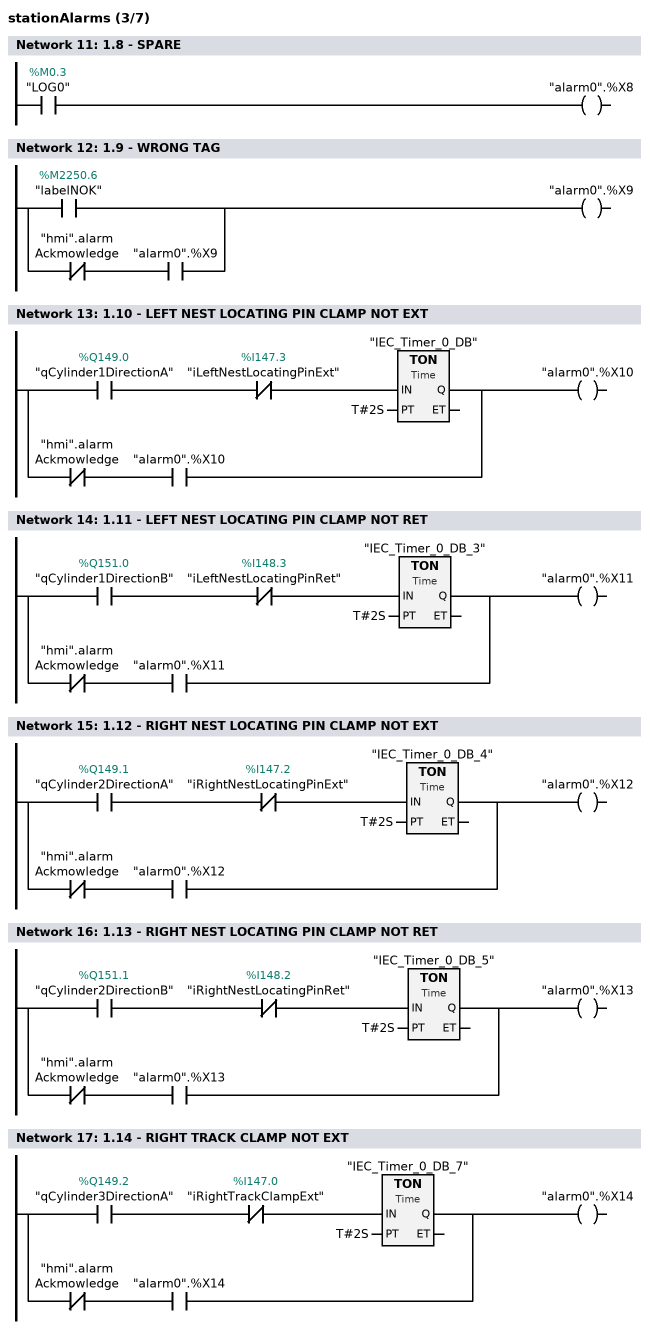
   RUNG wire#powerrail
      Contact( "LOG0" )
      Coil( "alarm0".%X8 )
   END_RUNG
   // the same network as SCL:
   "alarm0".%X8 := "LOG0";
END_REGION

REGION Network 12: 1.9 - WRONG TAG
   RUNG wire#powerrail
      Contact( "labelNOK" )
      wire#w1
      Coil( "alarm0".%X9 )
   END_RUNG
   RUNG wire#powerrail
      I_Contact( "hmi".alarmAckmowledge )
      Contact( "alarm0".%X9 )
   END_RUNG wire#w1
   // the same network as SCL:
   "alarm0".%X9 := "labelNOK" OR (NOT "hmi".alarmAckmowledge AND "alarm0".%X9);
END_REGION

REGION Network 13: 1.10 - LEFT NEST LOCATING PIN CLAMP NOT EXT
   RUNG wire#powerrail
      Contact( "qCylinder1DirectionA" )
      I_Contact( "iLeftNestLocatingPinExt" )
      { S7_Templates := "time_type := Time" } "IEC_Timer_0_DB".TON(pt := T#2S, et =>)
      wire#w1
      Coil( "alarm0".%X10 )
   END_RUNG
   RUNG wire#powerrail
      I_Contact( "hmi".alarmAckmowledge )
      Contact( "alarm0".%X10 )
   END_RUNG wire#w1
   // the same network as SCL:
   "IEC_Timer_0_DB".TON(IN := "qCylinder1DirectionA" AND NOT "iLeftNestLocatingPinExt", PT := T#2S);
   "alarm0".%X10 := "IEC_Timer_0_DB".Q OR (NOT "hmi".alarmAckmowledge AND "alarm0".%X10);
END_REGION

REGION Network 14: 1.11 - LEFT NEST LOCATING PIN CLAMP NOT RET
   RUNG wire#powerrail
      Contact( "qCylinder1DirectionB" )
      I_Contact( "iLeftNestLocatingPinRet" )
      { S7_Templates := "time_type := Time" } "IEC_Timer_0_DB_3".TON(pt := T#2S, et =>)
      wire#w1
      Coil( "alarm0".%X11 )
   END_RUNG
   RUNG wire#powerrail
      I_Contact( "hmi".alarmAckmowledge )
      Contact( "alarm0".%X11 )
   END_RUNG wire#w1
   // the same network as SCL:
   "IEC_Timer_0_DB_3".TON(IN := "qCylinder1DirectionB" AND NOT "iLeftNestLocatingPinRet", PT := T#2S);
   "alarm0".%X11 := "IEC_Timer_0_DB_3".Q OR (NOT "hmi".alarmAckmowledge AND "alarm0".%X11);
END_REGION

REGION Network 15: 1.12 - RIGHT NEST LOCATING PIN CLAMP NOT EXT
   RUNG wire#powerrail
      Contact( "qCylinder2DirectionA" )
      I_Contact( "iRightNestLocatingPinExt" )
      { S7_Templates := "time_type := Time" } "IEC_Timer_0_DB_4".TON(pt := T#2S, et =>)
      wire#w1
      Coil( "alarm0".%X12 )
   END_RUNG
   RUNG wire#powerrail
      I_Contact( "hmi".alarmAckmowledge )
      Contact( "alarm0".%X12 )
   END_RUNG wire#w1
   // the same network as SCL:
   "IEC_Timer_0_DB_4".TON(IN := "qCylinder2DirectionA" AND NOT "iRightNestLocatingPinExt", PT := T#2S);
   "alarm0".%X12 := "IEC_Timer_0_DB_4".Q OR (NOT "hmi".alarmAckmowledge AND "alarm0".%X12);
END_REGION

REGION Network 16: 1.13 - RIGHT NEST LOCATING PIN CLAMP NOT RET
   RUNG wire#powerrail
      Contact( "qCylinder2DirectionB" )
      I_Contact( "iRightNestLocatingPinRet" )
      { S7_Templates := "time_type := Time" } "IEC_Timer_0_DB_5".TON(pt := T#2S, et =>)
      wire#w1
      Coil( "alarm0".%X13 )
   END_RUNG
   RUNG wire#powerrail
      I_Contact( "hmi".alarmAckmowledge )
      Contact( "alarm0".%X13 )
   END_RUNG wire#w1
   // the same network as SCL:
   "IEC_Timer_0_DB_5".TON(IN := "qCylinder2DirectionB" AND NOT "iRightNestLocatingPinRet", PT := T#2S);
   "alarm0".%X13 := "IEC_Timer_0_DB_5".Q OR (NOT "hmi".alarmAckmowledge AND "alarm0".%X13);
END_REGION

REGION Network 17: 1.14 - RIGHT TRACK CLAMP NOT EXT
   RUNG wire#powerrail
      Contact( "qCylinder3DirectionA" )
      I_Contact( "iRightTrackClampExt" )
      { S7_Templates := "time_type := Time" } "IEC_Timer_0_DB_7".TON(pt := T#2S, et =>)
      wire#w1
      Coil( "alarm0".%X14 )
   END_RUNG
   RUNG wire#powerrail
      I_Contact( "hmi".alarmAckmowledge )
      Contact( "alarm0".%X14 )
   END_RUNG wire#w1
   // the same network as SCL:
   "IEC_Timer_0_DB_7".TON(IN := "qCylinder3DirectionA" AND NOT "iRightTrackClampExt", PT := T#2S);
   "alarm0".%X14 := "IEC_Timer_0_DB_7".Q OR (NOT "hmi".alarmAckmowledge AND "alarm0".%X14);
END_REGION

REGION Network 18: 1.15 - RIGHT TRACK CLAMP NOT RET
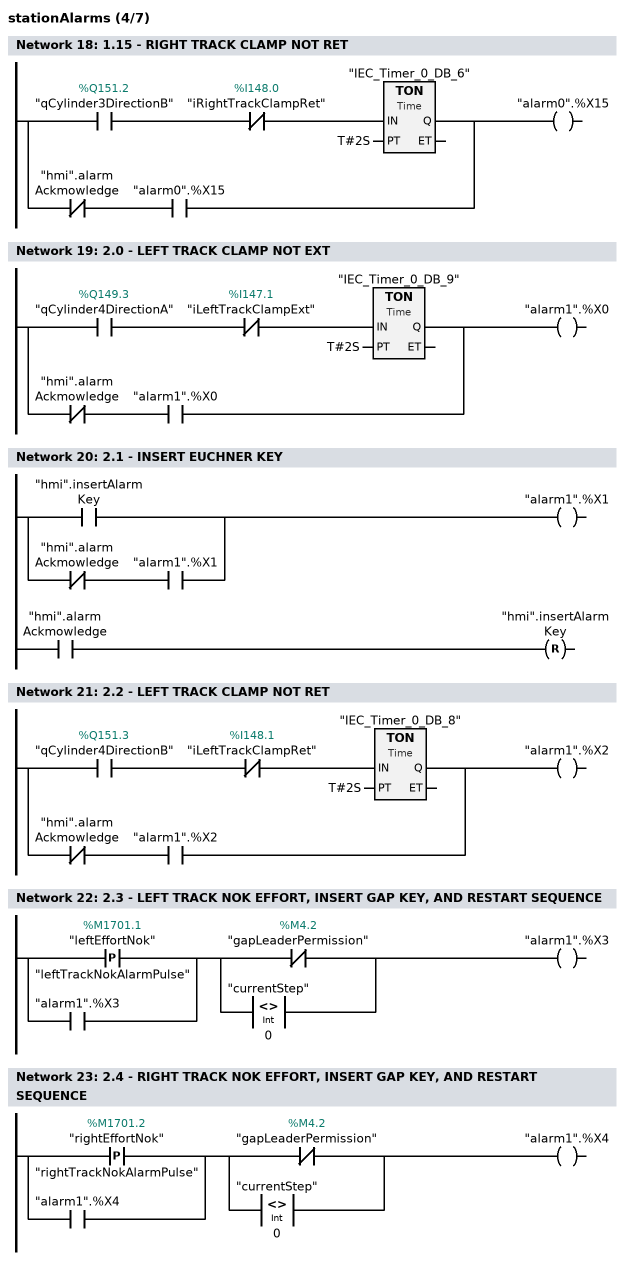
   RUNG wire#powerrail
      Contact( "qCylinder3DirectionB" )
      I_Contact( "iRightTrackClampRet" )
      { S7_Templates := "time_type := Time" } "IEC_Timer_0_DB_6".TON(pt := T#2S, et =>)
      wire#w1
      Coil( "alarm0".%X15 )
   END_RUNG
   RUNG wire#powerrail
      I_Contact( "hmi".alarmAckmowledge )
      Contact( "alarm0".%X15 )
   END_RUNG wire#w1
   // the same network as SCL:
   "IEC_Timer_0_DB_6".TON(IN := "qCylinder3DirectionB" AND NOT "iRightTrackClampRet", PT := T#2S);
   "alarm0".%X15 := "IEC_Timer_0_DB_6".Q OR (NOT "hmi".alarmAckmowledge AND "alarm0".%X15);
END_REGION

REGION Network 19: 2.0 - LEFT TRACK CLAMP NOT EXT
   RUNG wire#powerrail
      Contact( "qCylinder4DirectionA" )
      I_Contact( "iLeftTrackClampExt" )
      { S7_Templates := "time_type := Time" } "IEC_Timer_0_DB_9".TON(pt := T#2S, et =>)
      wire#w1
      Coil( "alarm1".%X0 )
   END_RUNG
   RUNG wire#powerrail
      I_Contact( "hmi".alarmAckmowledge )
      Contact( "alarm1".%X0 )
   END_RUNG wire#w1
   // the same network as SCL:
   "IEC_Timer_0_DB_9".TON(IN := "qCylinder4DirectionA" AND NOT "iLeftTrackClampExt", PT := T#2S);
   "alarm1".%X0 := "IEC_Timer_0_DB_9".Q OR (NOT "hmi".alarmAckmowledge AND "alarm1".%X0);
END_REGION

REGION Network 20: 2.1 - INSERT EUCHNER KEY
   RUNG wire#powerrail
      Contact( "hmi".insertAlarmKey )
      wire#w1
      Coil( "alarm1".%X1 )
   END_RUNG
   RUNG wire#powerrail
      I_Contact( "hmi".alarmAckmowledge )
      Contact( "alarm1".%X1 )
   END_RUNG wire#w1
   RUNG wire#powerrail
      Contact( "hmi".alarmAckmowledge )
      R_Coil( "hmi".insertAlarmKey )
   END_RUNG
   // the same network as SCL:
   "alarm1".%X1 := "hmi".insertAlarmKey OR (NOT "hmi".alarmAckmowledge AND "alarm1".%X1);
   IF "hmi".alarmAckmowledge THEN "hmi".insertAlarmKey := FALSE; END_IF;
END_REGION

REGION Network 21: 2.2 - LEFT TRACK CLAMP NOT RET
   RUNG wire#powerrail
      Contact( "qCylinder4DirectionB" )
      I_Contact( "iLeftTrackClampRet" )
      { S7_Templates := "time_type := Time" } "IEC_Timer_0_DB_8".TON(pt := T#2S, et =>)
      wire#w1
      Coil( "alarm1".%X2 )
   END_RUNG
   RUNG wire#powerrail
      I_Contact( "hmi".alarmAckmowledge )
      Contact( "alarm1".%X2 )
   END_RUNG wire#w1
   // the same network as SCL:
   "IEC_Timer_0_DB_8".TON(IN := "qCylinder4DirectionB" AND NOT "iLeftTrackClampRet", PT := T#2S);
   "alarm1".%X2 := "IEC_Timer_0_DB_8".Q OR (NOT "hmi".alarmAckmowledge AND "alarm1".%X2);
END_REGION

REGION Network 22: 2.3 - LEFT TRACK NOK EFFORT, INSERT GAP KEY, AND RESTART SEQUENCE
   RUNG wire#powerrail
      P_Contact(operand := "leftEffortNok", bit := "leftTrackNokAlarmPulse")
      wire#w1
      I_Contact( "gapLeaderPermission" )
      wire#w2
      Coil( "alarm1".%X3 )
   END_RUNG
   RUNG wire#powerrail
      Contact( "alarm1".%X3 )
   END_RUNG wire#w1
   RUNG wire#w1
      { S7_Templates := "SrcType := Int" } NE_Contact(in1 := "currentStep", in2 := 0)
   END_RUNG wire#w2
   // the same network as SCL:
   #_w1 := "leftEffortNok" AND NOT "leftTrackNokAlarmPulse";   // rising edge of "leftEffortNok"
   "leftTrackNokAlarmPulse" := "leftEffortNok";
   "alarm1".%X3 := (#_w1 OR "alarm1".%X3) AND (NOT "gapLeaderPermission" OR ("currentStep" <> 0));
END_REGION

REGION Network 23: 2.4 - RIGHT TRACK NOK EFFORT, INSERT GAP KEY, AND RESTART SEQUENCE
   RUNG wire#powerrail
      P_Contact(operand := "rightEffortNok", bit := "rightTrackNokAlarmPulse")
      wire#w1
      I_Contact( "gapLeaderPermission" )
      wire#w2
      Coil( "alarm1".%X4 )
   END_RUNG
   RUNG wire#powerrail
      Contact( "alarm1".%X4 )
   END_RUNG wire#w1
   RUNG wire#w1
      { S7_Templates := "SrcType := Int" } NE_Contact(in1 := "currentStep", in2 := 0)
   END_RUNG wire#w2
   // the same network as SCL:
   #_w1 := "rightEffortNok" AND NOT "rightTrackNokAlarmPulse";   // rising edge of "rightEffortNok"
   "rightTrackNokAlarmPulse" := "rightEffortNok";
   "alarm1".%X4 := (#_w1 OR "alarm1".%X4) AND (NOT "gapLeaderPermission" OR ("currentStep" <> 0));
END_REGION

REGION Network 24: 2.5 - SELECT MODELTO RUN
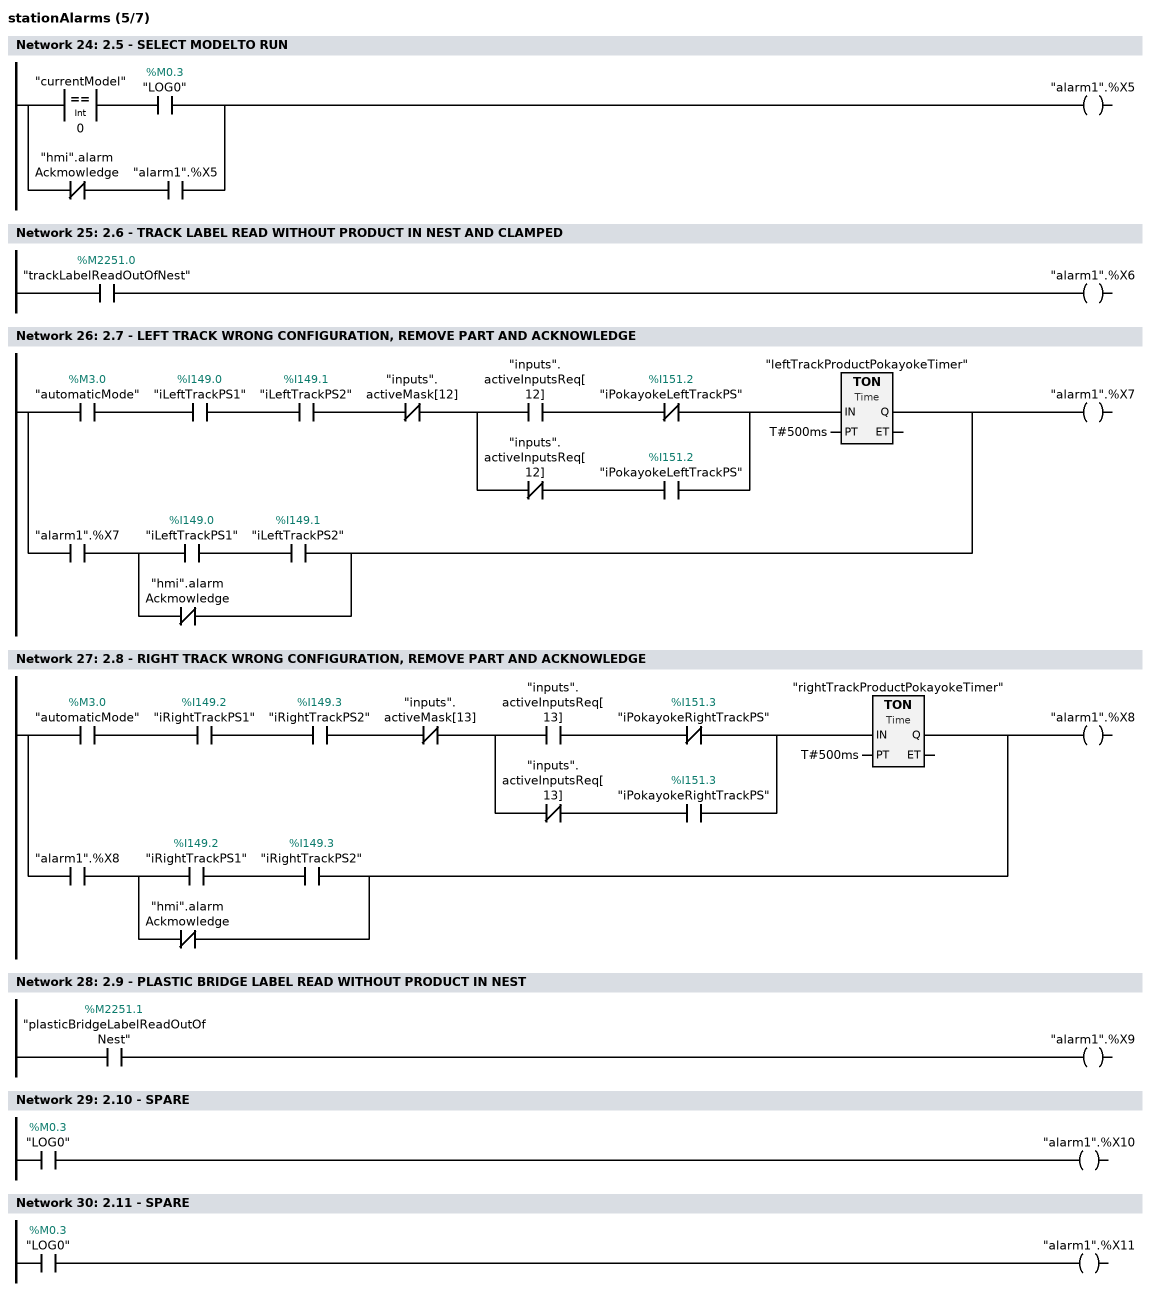
   RUNG wire#powerrail
      { S7_Templates := "SrcType := Int" } EQ_Contact(in1 := "currentModel", in2 := 0)
      Contact( "LOG0" )
      wire#w1
      Coil( "alarm1".%X5 )
   END_RUNG
   RUNG wire#powerrail
      I_Contact( "hmi".alarmAckmowledge )
      Contact( "alarm1".%X5 )
   END_RUNG wire#w1
   // the same network as SCL:
   "alarm1".%X5 := (("currentModel" = 0) AND "LOG0") OR (NOT "hmi".alarmAckmowledge AND "alarm1".%X5);
END_REGION

REGION Network 25: 2.6 - TRACK LABEL READ WITHOUT PRODUCT IN NEST AND CLAMPED
   RUNG wire#powerrail
      Contact( "trackLabelReadOutOfNest" )
      Coil( "alarm1".%X6 )
   END_RUNG
   // the same network as SCL:
   "alarm1".%X6 := "trackLabelReadOutOfNest";
END_REGION

REGION Network 26: 2.7 - LEFT TRACK WRONG CONFIGURATION, REMOVE PART AND ACKNOWLEDGE
   RUNG wire#powerrail
      Contact( "automaticMode" )
      Contact( "iLeftTrackPS1" )
      Contact( "iLeftTrackPS2" )
      I_Contact( "inputs".activeMask[12] )
      wire#w1
      Contact( "inputs".activeInputsReq[12] )
      I_Contact( "iPokayokeLeftTrackPS" )
      wire#w2
      { S7_Templates := "time_type := Time" } "leftTrackProductPokayokeTimer".TON(pt := T#500ms, et =>)
      wire#w3
      Coil( "alarm1".%X7 )
   END_RUNG
   RUNG wire#w1
      I_Contact( "inputs".activeInputsReq[12] )
      Contact( "iPokayokeLeftTrackPS" )
   END_RUNG wire#w2
   RUNG wire#powerrail
      Contact( "alarm1".%X7 )
      wire#w4
      Contact( "iLeftTrackPS1" )
      Contact( "iLeftTrackPS2" )
   END_RUNG wire#w3
   RUNG wire#w4
      I_Contact( "hmi".alarmAckmowledge )
   END_RUNG wire#w3
   // the same network as SCL:
   "leftTrackProductPokayokeTimer".TON(IN := "automaticMode" AND "iLeftTrackPS1" AND "iLeftTrackPS2" AND NOT "inputs".activeMask[12] AND (("inputs".activeInputsReq[12] AND NOT "iPokayokeLeftTrackPS") OR (NOT "inputs".activeInputsReq[12] AND "iPokayokeLeftTrackPS")),
                           PT := T#500ms);
   "alarm1".%X7 := "leftTrackProductPokayokeTimer".Q OR ("alarm1".%X7 AND (("iLeftTrackPS1" AND "iLeftTrackPS2") OR NOT "hmi".alarmAckmowledge));
END_REGION

REGION Network 27: 2.8 - RIGHT TRACK WRONG CONFIGURATION, REMOVE PART AND ACKNOWLEDGE
   RUNG wire#powerrail
      Contact( "automaticMode" )
      Contact( "iRightTrackPS1" )
      Contact( "iRightTrackPS2" )
      I_Contact( "inputs".activeMask[13] )
      wire#w1
      Contact( "inputs".activeInputsReq[13] )
      I_Contact( "iPokayokeRightTrackPS" )
      wire#w2
      { S7_Templates := "time_type := Time" } "rightTrackProductPokayokeTimer".TON(pt := T#500ms, et =>)
      wire#w3
      Coil( "alarm1".%X8 )
   END_RUNG
   RUNG wire#w1
      I_Contact( "inputs".activeInputsReq[13] )
      Contact( "iPokayokeRightTrackPS" )
   END_RUNG wire#w2
   RUNG wire#powerrail
      Contact( "alarm1".%X8 )
      wire#w4
      Contact( "iRightTrackPS1" )
      Contact( "iRightTrackPS2" )
   END_RUNG wire#w3
   RUNG wire#w4
      I_Contact( "hmi".alarmAckmowledge )
   END_RUNG wire#w3
   // the same network as SCL:
   "rightTrackProductPokayokeTimer".TON(IN := "automaticMode" AND "iRightTrackPS1" AND "iRightTrackPS2" AND NOT "inputs".activeMask[13] AND (("inputs".activeInputsReq[13] AND NOT "iPokayokeRightTrackPS") OR (NOT "inputs".activeInputsReq[13] AND "iPokayokeRightTrackPS")),
                           PT := T#500ms);
   "alarm1".%X8 := "rightTrackProductPokayokeTimer".Q OR ("alarm1".%X8 AND (("iRightTrackPS1" AND "iRightTrackPS2") OR NOT "hmi".alarmAckmowledge));
END_REGION

REGION Network 28: 2.9 - PLASTIC BRIDGE LABEL READ WITHOUT PRODUCT IN NEST
   RUNG wire#powerrail
      Contact( "plasticBridgeLabelReadOutOfNest" )
      Coil( "alarm1".%X9 )
   END_RUNG
   // the same network as SCL:
   "alarm1".%X9 := "plasticBridgeLabelReadOutOfNest";
END_REGION

REGION Network 29: 2.10 - SPARE
   RUNG wire#powerrail
      Contact( "LOG0" )
      Coil( "alarm1".%X10 )
   END_RUNG
   // the same network as SCL:
   "alarm1".%X10 := "LOG0";
END_REGION

REGION Network 30: 2.11 - SPARE
   RUNG wire#powerrail
      Contact( "LOG0" )
      Coil( "alarm1".%X11 )
   END_RUNG
   // the same network as SCL:
   "alarm1".%X11 := "LOG0";
END_REGION

REGION Network 31: 2.12 INSERT KEY TO LIBERATE
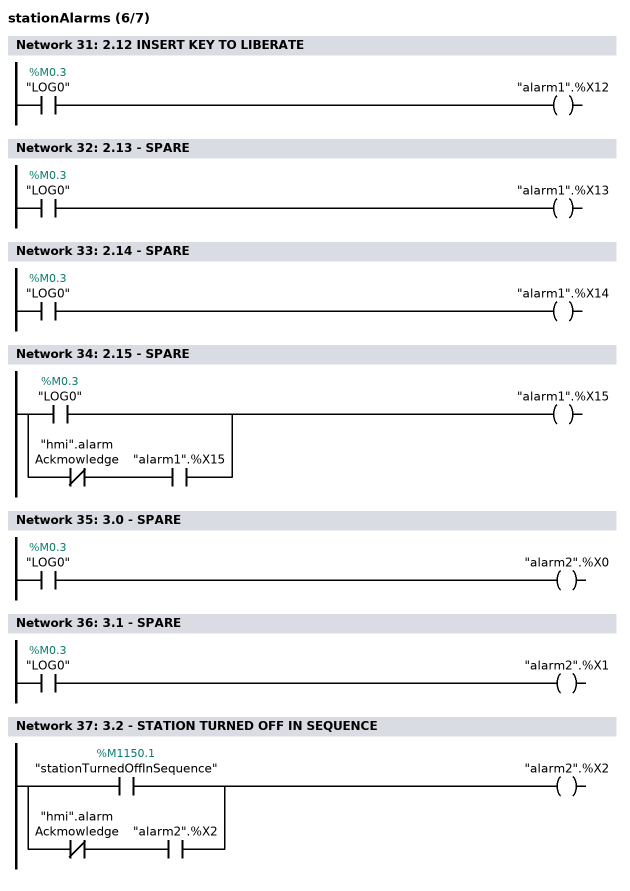
   RUNG wire#powerrail
      Contact( "LOG0" )
      Coil( "alarm1".%X12 )
   END_RUNG
   // the same network as SCL:
   "alarm1".%X12 := "LOG0";
END_REGION

REGION Network 32: 2.13 - SPARE
   RUNG wire#powerrail
      Contact( "LOG0" )
      Coil( "alarm1".%X13 )
   END_RUNG
   // the same network as SCL:
   "alarm1".%X13 := "LOG0";
END_REGION

REGION Network 33: 2.14 - SPARE
   RUNG wire#powerrail
      Contact( "LOG0" )
      Coil( "alarm1".%X14 )
   END_RUNG
   // the same network as SCL:
   "alarm1".%X14 := "LOG0";
END_REGION

REGION Network 34: 2.15 - SPARE
   RUNG wire#powerrail
      Contact( "LOG0" )
      wire#w1
      Coil( "alarm1".%X15 )
   END_RUNG
   RUNG wire#powerrail
      I_Contact( "hmi".alarmAckmowledge )
      Contact( "alarm1".%X15 )
   END_RUNG wire#w1
   // the same network as SCL:
   "alarm1".%X15 := "LOG0" OR (NOT "hmi".alarmAckmowledge AND "alarm1".%X15);
END_REGION

REGION Network 35: 3.0 - SPARE
   RUNG wire#powerrail
      Contact( "LOG0" )
      Coil( "alarm2".%X0 )
   END_RUNG
   // the same network as SCL:
   "alarm2".%X0 := "LOG0";
END_REGION

REGION Network 36: 3.1 - SPARE
   RUNG wire#powerrail
      Contact( "LOG0" )
      Coil( "alarm2".%X1 )
   END_RUNG
   // the same network as SCL:
   "alarm2".%X1 := "LOG0";
END_REGION

REGION Network 37: 3.2 - STATION TURNED OFF IN SEQUENCE
   RUNG wire#powerrail
      Contact( "stationTurnedOffInSequence" )
      wire#w1
      Coil( "alarm2".%X2 )
   END_RUNG
   RUNG wire#powerrail
      I_Contact( "hmi".alarmAckmowledge )
      Contact( "alarm2".%X2 )
   END_RUNG wire#w1
   // the same network as SCL:
   "alarm2".%X2 := "stationTurnedOffInSequence" OR (NOT "hmi".alarmAckmowledge AND "alarm2".%X2);
END_REGION

REGION Network 38: 3.3 - 3.13 COMMUNICATION ALARMS
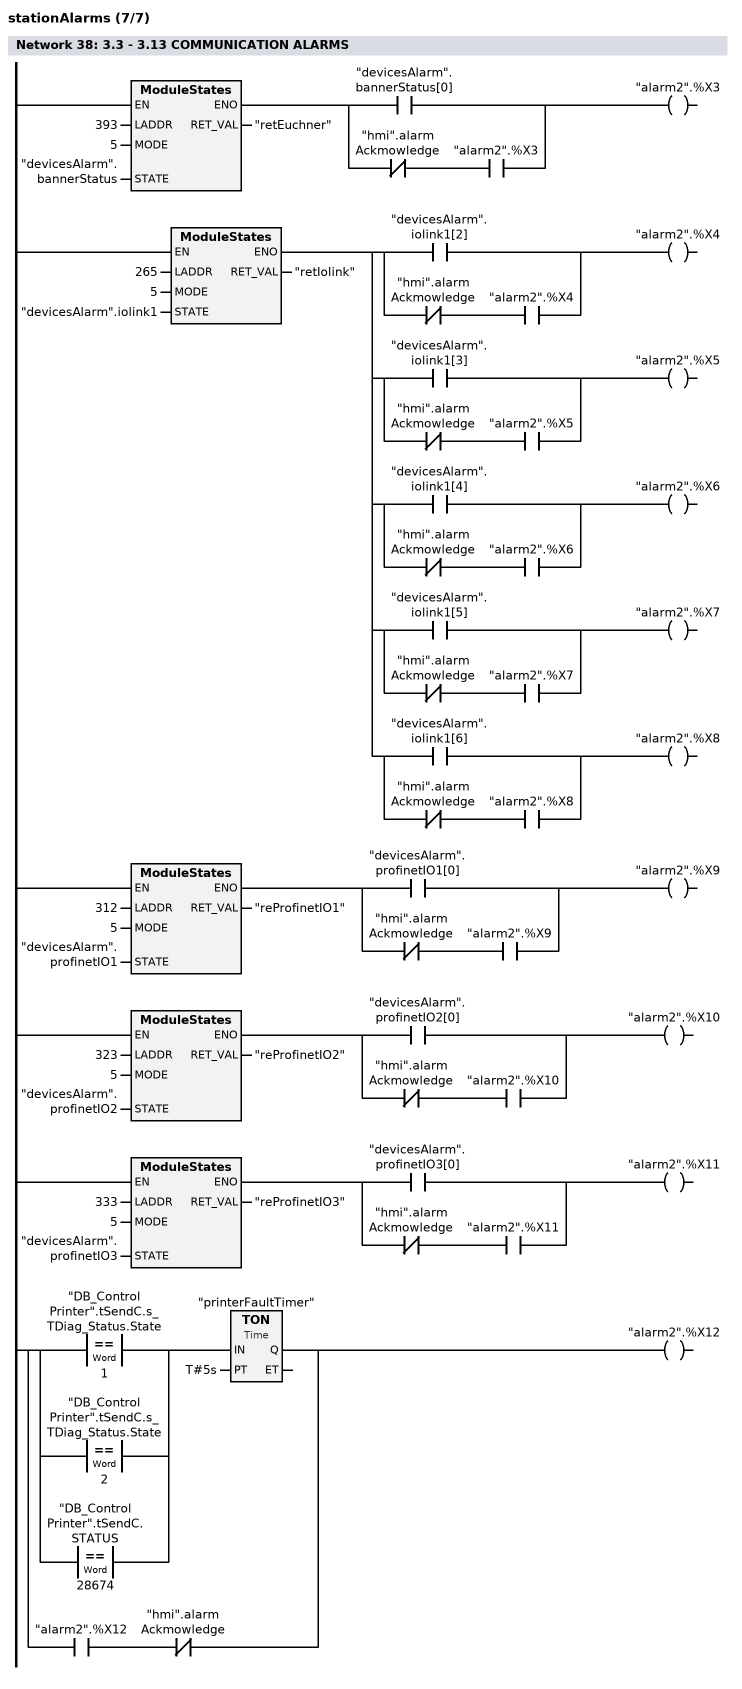
   RUNG wire#powerrail
      ModuleStates(LADDR := 393, MODE := 5, STATE := "devicesAlarm".bannerStatus, Ret_Val => "retEuchner")
      wire#w1
      Contact( "devicesAlarm".bannerStatus[0] )
      wire#w2
      Coil( "alarm2".%X3 )
   END_RUNG
   RUNG wire#w1
      I_Contact( "hmi".alarmAckmowledge )
      Contact( "alarm2".%X3 )
   END_RUNG wire#w2
   RUNG wire#powerrail
      ModuleStates(LADDR := 265, MODE := 5, STATE := "devicesAlarm".iolink1, Ret_Val => "retIolink")
      wire#w3
      Contact( "devicesAlarm".iolink1[2] )
      wire#w4
      Coil( "alarm2".%X4 )
   END_RUNG
   RUNG wire#w3
      I_Contact( "hmi".alarmAckmowledge )
      Contact( "alarm2".%X4 )
   END_RUNG wire#w4
   RUNG wire#w3
      Contact( "devicesAlarm".iolink1[3] )
      wire#w5
      Coil( "alarm2".%X5 )
   END_RUNG
   RUNG wire#w3
      I_Contact( "hmi".alarmAckmowledge )
      Contact( "alarm2".%X5 )
   END_RUNG wire#w5
   RUNG wire#w3
      Contact( "devicesAlarm".iolink1[4] )
      wire#w6
      Coil( "alarm2".%X6 )
   END_RUNG
   RUNG wire#w3
      I_Contact( "hmi".alarmAckmowledge )
      Contact( "alarm2".%X6 )
   END_RUNG wire#w6
   RUNG wire#w3
      Contact( "devicesAlarm".iolink1[5] )
      wire#w7
      Coil( "alarm2".%X7 )
   END_RUNG
   RUNG wire#w3
      I_Contact( "hmi".alarmAckmowledge )
      Contact( "alarm2".%X7 )
   END_RUNG wire#w7
   RUNG wire#w3
      Contact( "devicesAlarm".iolink1[6] )
      wire#w8
      Coil( "alarm2".%X8 )
   END_RUNG
   RUNG wire#w3
      I_Contact( "hmi".alarmAckmowledge )
      Contact( "alarm2".%X8 )
   END_RUNG wire#w8
   RUNG wire#powerrail
      ModuleStates(LADDR := 312, MODE := 5, STATE := "devicesAlarm".profinetIO1, Ret_Val => "reProfinetIO1")
      wire#w9
      Contact( "devicesAlarm".profinetIO1[0] )
      wire#w10
      Coil( "alarm2".%X9 )
   END_RUNG
   RUNG wire#w9
      I_Contact( "hmi".alarmAckmowledge )
      Contact( "alarm2".%X9 )
   END_RUNG wire#w10
   RUNG wire#powerrail
      ModuleStates(LADDR := 323, MODE := 5, STATE := "devicesAlarm".profinetIO2, Ret_Val => "reProfinetIO2")
      wire#w11
      Contact( "devicesAlarm".profinetIO2[0] )
      wire#w12
      Coil( "alarm2".%X10 )
   END_RUNG
   RUNG wire#w11
      I_Contact( "hmi".alarmAckmowledge )
      Contact( "alarm2".%X10 )
   END_RUNG wire#w12
   RUNG wire#powerrail
      ModuleStates(LADDR := 333, MODE := 5, STATE := "devicesAlarm".profinetIO3, Ret_Val => "reProfinetIO3")
      wire#w13
      Contact( "devicesAlarm".profinetIO3[0] )
      wire#w14
      Coil( "alarm2".%X11 )
   END_RUNG
   RUNG wire#w13
      I_Contact( "hmi".alarmAckmowledge )
      Contact( "alarm2".%X11 )
   END_RUNG wire#w14
   RUNG wire#powerrail
      { S7_Templates := "SrcType := Word" } EQ_Contact(in1 := "DB_ControlPrinter".tSendC.s_TDiag_Status.State, in2 := 1)
      wire#w15
      { S7_Templates := "time_type := Time" } "printerFaultTimer".TON(pt := T#5s, et =>)
      wire#w16
      Coil( "alarm2".%X12 )
   END_RUNG
   RUNG wire#powerrail
      { S7_Templates := "SrcType := Word" } EQ_Contact(in1 := "DB_ControlPrinter".tSendC.s_TDiag_Status.State, in2 := 2)
   END_RUNG wire#w15
   RUNG wire#powerrail
      { S7_Templates := "SrcType := Word" } EQ_Contact(in1 := "DB_ControlPrinter".tSendC.STATUS, in2 := 28674)
   END_RUNG wire#w15
   RUNG wire#powerrail
      Contact( "alarm2".%X12 )
      I_Contact( "hmi".alarmAckmowledge )
   END_RUNG wire#w16
   // the same network as SCL:
   "retEuchner" := ModuleStates(LADDR := 393, MODE := 5, STATE := "devicesAlarm".bannerStatus, ENO => #_w1);
   "alarm2".%X3 := #_w1 AND ("devicesAlarm".bannerStatus[0] OR (NOT "hmi".alarmAckmowledge AND "alarm2".%X3));
   "retIolink" := ModuleStates(LADDR := 265, MODE := 5, STATE := "devicesAlarm".iolink1, ENO => #_w2);
   "alarm2".%X4 := #_w2 AND ("devicesAlarm".iolink1[2] OR (NOT "hmi".alarmAckmowledge AND "alarm2".%X4));
   "alarm2".%X5 := #_w2 AND ("devicesAlarm".iolink1[3] OR (NOT "hmi".alarmAckmowledge AND "alarm2".%X5));
   "alarm2".%X6 := #_w2 AND ("devicesAlarm".iolink1[4] OR (NOT "hmi".alarmAckmowledge AND "alarm2".%X6));
   "alarm2".%X7 := #_w2 AND ("devicesAlarm".iolink1[5] OR (NOT "hmi".alarmAckmowledge AND "alarm2".%X7));
   "alarm2".%X8 := #_w2 AND ("devicesAlarm".iolink1[6] OR (NOT "hmi".alarmAckmowledge AND "alarm2".%X8));
   "reProfinetIO1" := ModuleStates(LADDR := 312, MODE := 5, STATE := "devicesAlarm".profinetIO1, ENO => #_w3);
   "alarm2".%X9 := #_w3 AND ("devicesAlarm".profinetIO1[0] OR (NOT "hmi".alarmAckmowledge AND "alarm2".%X9));
   "reProfinetIO2" := ModuleStates(LADDR := 323, MODE := 5, STATE := "devicesAlarm".profinetIO2, ENO => #_w4);
   "alarm2".%X10 := #_w4 AND ("devicesAlarm".profinetIO2[0] OR (NOT "hmi".alarmAckmowledge AND "alarm2".%X10));
   "reProfinetIO3" := ModuleStates(LADDR := 333, MODE := 5, STATE := "devicesAlarm".profinetIO3, ENO => #_w5);
   "alarm2".%X11 := #_w5 AND ("devicesAlarm".profinetIO3[0] OR (NOT "hmi".alarmAckmowledge AND "alarm2".%X11));
   "printerFaultTimer".TON(IN := ("DB_ControlPrinter".tSendC.s_TDiag_Status.State = 1) OR ("DB_ControlPrinter".tSendC.s_TDiag_Status.State = 2) OR ("DB_ControlPrinter".tSendC.STATUS = 28674),
                           PT := T#5s);
   "alarm2".%X12 := "printerFaultTimer".Q OR ("alarm2".%X12 AND NOT "hmi".alarmAckmowledge);
END_REGION
END_FUNCTION

FUNCTION_BLOCK "timeSystem"   // FB2420, LAD
{ S7_Optimized_Access := 'TRUE' }
VERSION : 0.1
// stored: AutoNumber false, IsIECCheckEnabled false, IsRetainMemResEnabled false, MemoryReserve 100, SetENOAutomatically false, UDAEnableTagReadback false
   VAR_INPUT
      bPartOkNok : Bool;
      bRunningcycle : Bool;
      bPreCount : Bool;
   END_VAR
   VAR_OUTPUT
      bShift1 : Bool;
      bShift2 : Bool;
      bShift3 : Bool;
      nCycle_Time_Shift : Real;
      nCycleTimeAvg_Shift1 : Real;
      nCycleTimeAvg_Shift2 : Real;
      nCycleTimeAvg_Shift3 : Real;
   END_VAR
   VAR
      Ret_Val_WR { ExternalAccessible := 'False'; ExternalVisible := 'False'; ExternalWritable := 'False'} : USInt;
      Ret_Val_RD { ExternalAccessible := 'False'; ExternalVisible := 'False'; ExternalWritable := 'False'} : USInt;
      DTL_Set_Time : DTL;
      DTL_Read_Time : DTL;
      TOD_Read : Time_Of_Day;
      Date_Read : Date;
      bAceptButtonHmiP : Bool;
      bAcept_buttonHMI : Bool;
      nSet_minute : Int;
      nSet_Hour : Int;
      nSet_Day : Int;
      nSet_Month : Int;
      nSet_Year : Int;
      nCycleTimeArray : Array[0..5] of Real;
      tCycleTime { S7_SetPoint := 'True'} : IEC_TIMER;
      nCycleTimeET : UDInt;
      tCycleTimeTotal : UDInt;
      bPartOkNokP : Bool;
      bPartOkNokCmd : Bool;
      nPartAvgCounter : Int;
      bCycle_StartedP : Bool;
      bSH1 : Bool;
      bSH2 : Bool;
      bSH3 : Bool;
      nCycle_Time : Real;
      nCycleTimeAvg : Real;
      Read_Local_Time : DTL;
      Read_System_Time : DTL;
      Time_HMI_Set : DTL;
      RetVal1 : Word;
      Retval2 : Word;
      Retval3 : Word;
      n : Int;
      timesCounter { S7_SetPoint := 'True'} : IEC_COUNTER;
   END_VAR
   VAR RETAIN
      tCycle_Running : Real;
   END_VAR
   VAR
      nCycleAvg : DInt;
      nCycleTime_Total : Time_Of_Day;
      ntimeRun_conv : UDInt;
   END_VAR
   // nCycleTimeArray[3..5] := 0.0;
   VAR_TEMP   // added for the SCL form of the ladder/FBD networks
      _w1 : Bool;
   END_VAR
BEGIN

REGION Network 1: SET HOUR
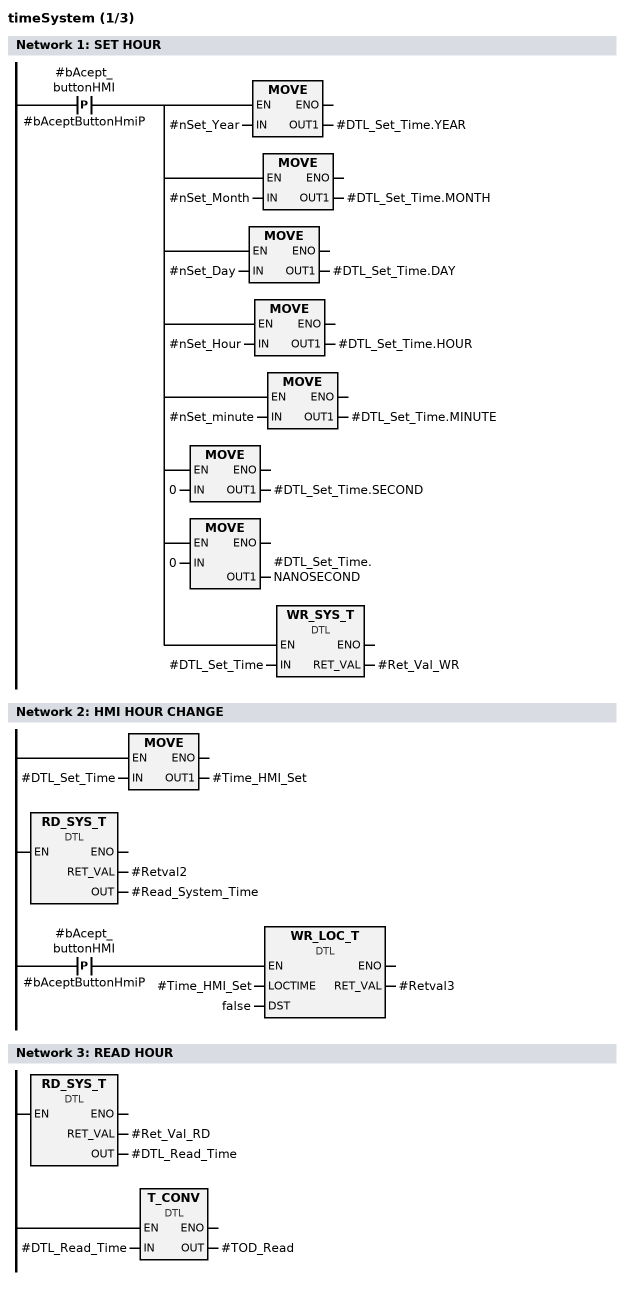
   RUNG wire#powerrail
      P_Contact(operand := #bAcept_buttonHMI, bit := #bAceptButtonHmiP)
      wire#w1
      Move(in := #nSet_Year, out1 => #DTL_Set_Time.YEAR)
   END_RUNG
   RUNG wire#w1
      Move(in := #nSet_Month, out1 => #DTL_Set_Time.MONTH)
   END_RUNG
   RUNG wire#w1
      Move(in := #nSet_Day, out1 => #DTL_Set_Time.DAY)
   END_RUNG
   RUNG wire#w1
      Move(in := #nSet_Hour, out1 => #DTL_Set_Time.HOUR)
   END_RUNG
   RUNG wire#w1
      Move(in := #nSet_minute, out1 => #DTL_Set_Time.MINUTE)
   END_RUNG
   RUNG wire#w1
      Move(in := 0, out1 => #DTL_Set_Time.SECOND)
   END_RUNG
   RUNG wire#w1
      Move(in := 0, out1 => #DTL_Set_Time.NANOSECOND)
   END_RUNG
   RUNG wire#w1
      { S7_Templates := "date_type := DTL" } WR_SYS_T(IN := #DTL_Set_Time, RET_VAL => #Ret_Val_WR)
   END_RUNG
   // the same network as SCL:
   #_w1 := #bAcept_buttonHMI AND NOT #bAceptButtonHmiP;   // rising edge of #bAcept_buttonHMI
   #bAceptButtonHmiP := #bAcept_buttonHMI;
   IF #_w1 THEN
       #DTL_Set_Time.YEAR := #nSet_Year;
       #DTL_Set_Time.MONTH := #nSet_Month;
       #DTL_Set_Time.DAY := #nSet_Day;
       #DTL_Set_Time.HOUR := #nSet_Hour;
       #DTL_Set_Time.MINUTE := #nSet_minute;
       #DTL_Set_Time.SECOND := 0;
       #DTL_Set_Time.NANOSECOND := 0;
       #Ret_Val_WR := WR_SYS_T(IN := #DTL_Set_Time);
   END_IF;
END_REGION

REGION Network 2: HMI HOUR CHANGE
   RUNG wire#powerrail
      Move(in := #DTL_Set_Time, out1 => #Time_HMI_Set)
   END_RUNG
   RUNG wire#powerrail
      { S7_Templates := "date_type := DTL" } RD_SYS_T(RET_VAL => #Retval2, OUT => #Read_System_Time)
   END_RUNG
   RUNG wire#powerrail
      P_Contact(operand := #bAcept_buttonHMI, bit := #bAceptButtonHmiP)
      { S7_Templates := "loctime_type := DTL" } WR_LOC_T(LOCTIME := #Time_HMI_Set, DST := false, Ret_Val => #Retval3)
   END_RUNG
   // the same network as SCL:
   #Time_HMI_Set := #DTL_Set_Time;
   #Retval2 := RD_SYS_T(OUT => #Read_System_Time);
   #_w1 := #bAcept_buttonHMI AND NOT #bAceptButtonHmiP;   // rising edge of #bAcept_buttonHMI
   #bAceptButtonHmiP := #bAcept_buttonHMI;
   IF #_w1 THEN #Retval3 := WR_LOC_T(LOCTIME := #Time_HMI_Set, DST := false); END_IF;
END_REGION

REGION Network 3: READ HOUR
   RUNG wire#powerrail
      { S7_Templates := "date_type := DTL" } RD_SYS_T(RET_VAL => #Ret_Val_RD, OUT => #DTL_Read_Time)
   END_RUNG
   RUNG wire#powerrail
      { S7_Templates := "[src_type := DTL, dest_type := Time_Of_Day]" } T_CONV(IN := #DTL_Read_Time, OUT => #TOD_Read)
   END_RUNG
   // the same network as SCL:
   #Ret_Val_RD := RD_SYS_T(OUT => #DTL_Read_Time);
   T_CONV(IN := #DTL_Read_Time, OUT => #TOD_Read);
END_REGION

REGION Network 4: WORK SHIFTS
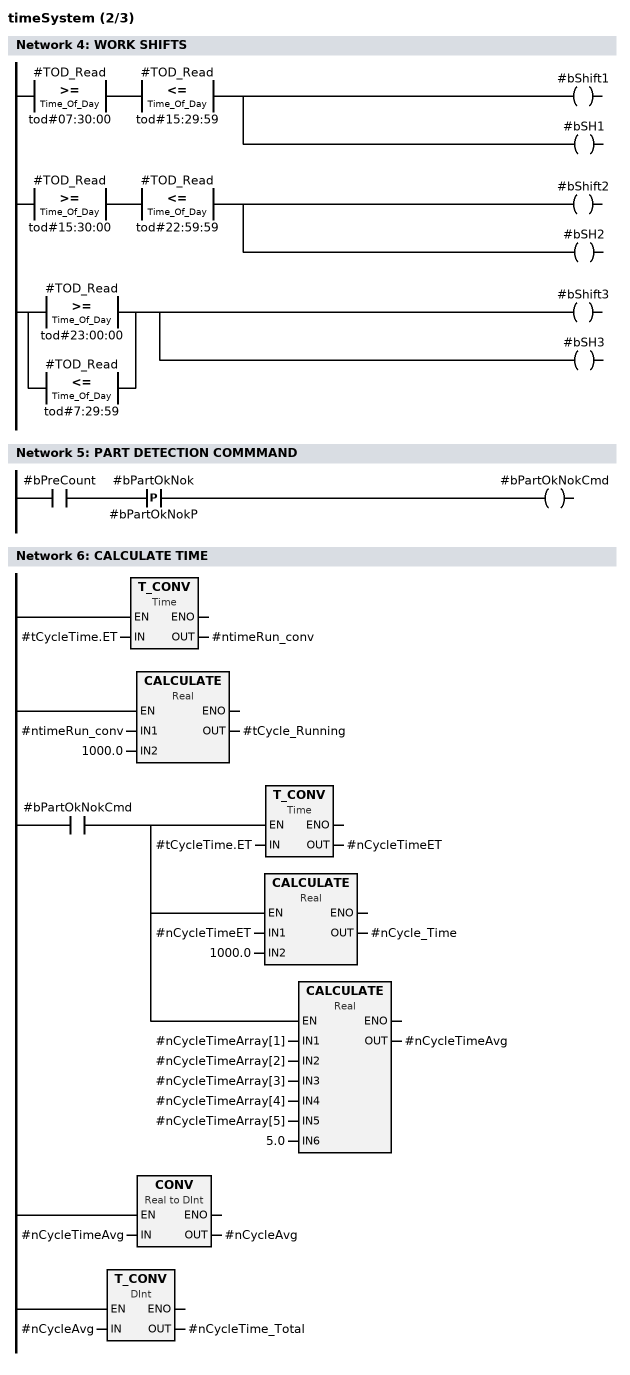
   RUNG wire#powerrail
      { S7_Templates := "SrcType := Time_Of_Day" } GE_Contact(in1 := #TOD_Read, in2 := tod#07:30:00)
      { S7_Templates := "SrcType := Time_Of_Day" } LE_Contact(in1 := #TOD_Read, in2 := tod#15:29:59)
      wire#w1
      Coil( #bShift1 )
   END_RUNG
   RUNG wire#w1
      Coil( #bSH1 )
   END_RUNG
   RUNG wire#powerrail
      { S7_Templates := "SrcType := Time_Of_Day" } GE_Contact(in1 := #TOD_Read, in2 := tod#15:30:00)
      { S7_Templates := "SrcType := Time_Of_Day" } LE_Contact(in1 := #TOD_Read, in2 := tod#22:59:59)
      wire#w2
      Coil( #bShift2 )
   END_RUNG
   RUNG wire#w2
      Coil( #bSH2 )
   END_RUNG
   RUNG wire#powerrail
      { S7_Templates := "SrcType := Time_Of_Day" } GE_Contact(in1 := #TOD_Read, in2 := tod#23:00:00)
      wire#w3
      Coil( #bShift3 )
   END_RUNG
   RUNG wire#powerrail
      { S7_Templates := "SrcType := Time_Of_Day" } LE_Contact(in1 := #TOD_Read, in2 := tod#7:29:59)
   END_RUNG wire#w3
   RUNG wire#w3
      Coil( #bSH3 )
   END_RUNG
   // the same network as SCL:
   #bShift1 := (#TOD_Read >= tod#07:30:00) AND (#TOD_Read <= tod#15:29:59);
   #bSH1 := #bShift1;
   #bShift2 := (#TOD_Read >= tod#15:30:00) AND (#TOD_Read <= tod#22:59:59);
   #bSH2 := #bShift2;
   #bShift3 := (#TOD_Read >= tod#23:00:00) OR (#TOD_Read <= tod#7:29:59);
   #bSH3 := #bShift3;
END_REGION

REGION Network 5: PART DETECTION COMMMAND
   RUNG wire#powerrail
      Contact( #bPreCount )
      P_Contact(operand := #bPartOkNok, bit := #bPartOkNokP)
      Coil( #bPartOkNokCmd )
   END_RUNG
   // the same network as SCL:
   #_w1 := #bPreCount AND #bPartOkNok AND NOT #bPartOkNokP;   // rising edge of #bPartOkNok
   #bPartOkNokP := #bPartOkNok;
   #bPartOkNokCmd := #_w1;
END_REGION

REGION Network 6: CALCULATE TIME
   RUNG wire#powerrail
      { S7_Templates := "[src_type := Time, dest_type := UDInt]" } T_CONV(IN := #tCycleTime.ET, OUT => #ntimeRun_conv)
   END_RUNG
   RUNG wire#powerrail
      { S7_Templates := "SrcType := Real"; S7_Expression := "in1/in2" } Calculate(in1 := #ntimeRun_conv, in2 := 1000.0, out => #tCycle_Running)
   END_RUNG
   RUNG wire#powerrail
      Contact( #bPartOkNokCmd )
      wire#w1
      { S7_Templates := "[src_type := Time, dest_type := UDInt]" } T_CONV(IN := #tCycleTime.ET, OUT => #nCycleTimeET)
   END_RUNG
   RUNG wire#w1
      { S7_Templates := "SrcType := Real"; S7_Expression := "in1/in2" } Calculate(in1 := #nCycleTimeET, in2 := 1000.0, out => #nCycle_Time)
   END_RUNG
   RUNG wire#w1
      { S7_Templates := "SrcType := Real"; S7_Expression := "(in1+in2+in3+in4+in5)/in6" } Calculate(in1 := #nCycleTimeArray[1], in2 := #nCycleTimeArray[2], in3 := #nCycleTimeArray[3], in4 := #nCycleTimeArray[4], in5 := #nCycleTimeArray[5], in6 := 5.0, out => #nCycleTimeAvg)
   END_RUNG
   RUNG wire#powerrail
      { S7_Templates := "[SrcType := Real, DestType := DInt]" } Convert(in := #nCycleTimeAvg, out => #nCycleAvg)
   END_RUNG
   RUNG wire#powerrail
      { S7_Templates := "[src_type := DInt, dest_type := Time_Of_Day]" } T_CONV(IN := #nCycleAvg, OUT => #nCycleTime_Total)
   END_RUNG
   // the same network as SCL:
   T_CONV(IN := #tCycleTime.ET, OUT => #ntimeRun_conv);
   #tCycle_Running := #ntimeRun_conv/1000.0;
   IF #bPartOkNokCmd THEN
       T_CONV(IN := #tCycleTime.ET, OUT => #nCycleTimeET);
       #nCycle_Time := #nCycleTimeET/1000.0;
       #nCycleTimeAvg := (#nCycleTimeArray[1]+#nCycleTimeArray[2]+#nCycleTimeArray[3]+#nCycleTimeArray[4]+#nCycleTimeArray[5])/5.0;
   END_IF;
   #nCycleAvg := REAL_TO_DINT(#nCycleTimeAvg);
   T_CONV(IN := #nCycleAvg, OUT => #nCycleTime_Total);
END_REGION

REGION Network 7: CICLE TIME ARRANGEMENT
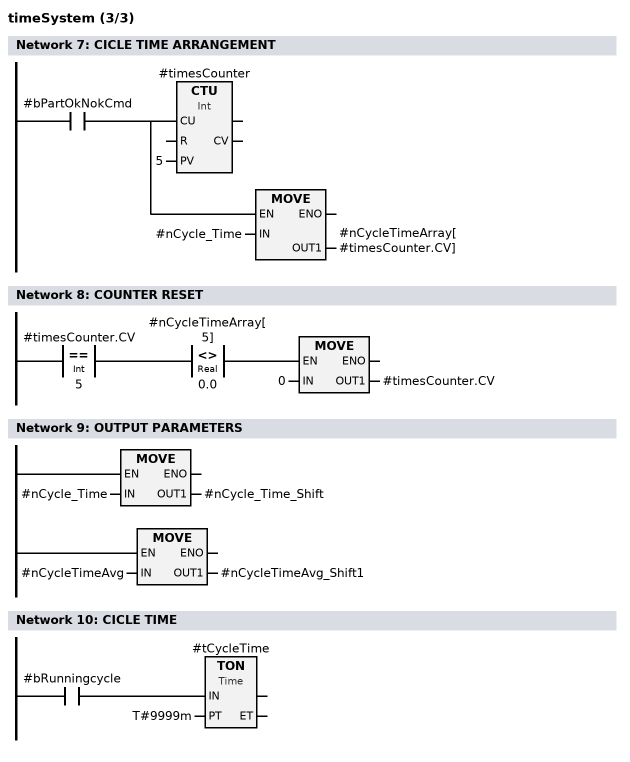
   RUNG wire#powerrail
      Contact( #bPartOkNokCmd )
      wire#w1
      { S7_Templates := "value_type := Int" } #timesCounter.CTU(r :=, pv := 5, cv =>)
   END_RUNG
   RUNG wire#w1
      Move(in := #nCycle_Time, out1 => #nCycleTimeArray[#timesCounter.CV])
   END_RUNG
   // the same network as SCL:
   #timesCounter.CTU(CU := #bPartOkNokCmd, PV := 5);
   IF #bPartOkNokCmd THEN #nCycleTimeArray[#timesCounter.CV] := #nCycle_Time; END_IF;
END_REGION

REGION Network 8: COUNTER RESET
   RUNG wire#powerrail
      { S7_Templates := "SrcType := Int" } EQ_Contact(in1 := #timesCounter.CV, in2 := 5)
      { S7_Templates := "SrcType := Real" } NE_Contact(in1 := #nCycleTimeArray[5], in2 := 0.0)
      Move(in := 0, out1 => #timesCounter.CV)
   END_RUNG
   // the same network as SCL:
   IF (#timesCounter.CV = 5) AND (#nCycleTimeArray[5] <> 0.0) THEN #timesCounter.CV := 0; END_IF;
END_REGION

REGION Network 9: OUTPUT PARAMETERS
   RUNG wire#powerrail
      Move(in := #nCycle_Time, out1 => #nCycle_Time_Shift)
   END_RUNG
   RUNG wire#powerrail
      Move(in := #nCycleTimeAvg, out1 => #nCycleTimeAvg_Shift1)
   END_RUNG
   // the same network as SCL:
   #nCycle_Time_Shift := #nCycle_Time;
   #nCycleTimeAvg_Shift1 := #nCycleTimeAvg;
END_REGION

REGION Network 10: CICLE TIME
   RUNG wire#powerrail
      Contact( #bRunningcycle )
      { S7_Templates := "time_type := Time" } #tCycleTime.TON(pt := T#9999m, et =>)
   END_RUNG
   // the same network as SCL:
   #tCycleTime.TON(IN := #bRunningcycle, PT := T#9999m);
END_REGION
END_FUNCTION_BLOCK

FUNCTION "eksFC" : Void   // FC305, LAD
TITLE = Euchner Management EKS KEY
{ S7_Optimized_Access := 'FALSE' }
VERSION : 0.1
// stored: AutoNumber false, IsIECCheckEnabled false, SetENOAutomatically false, UDAEnableTagReadback false
   VAR_INPUT
      iKeyIn : Bool;
      iEksLevel : Byte;
      iEksEmployeeID : DWord;
      iEksKeyID1 : DWord;
      iEksKeyID2 : DWord;
      iEksJobFinished : Bool;
      hmiCurrentPage : Word;
   END_VAR
   VAR_OUTPUT
      qEksStartAdress : Byte;
      qEksDataLength : Byte;
      qEksData1 : Byte;
      qEksData2 : DWord;
      qEksWriteCommand : Bool;
   END_VAR
   VAR_TEMP
      tNone : Bool;
      tDBAddressKeys : Int;
      tDBAddressHMIPage : Int;
      tDBKeyStructLength : Int;
      tDBAddress : Int;
      tDBLength : Int;
      tCycle : Int;
      tFill : Int;
      tKey : "udt_EKS_KEY";
      tDBStartAddress : Int;
      tsearch : Bool;
      i : Int;
   END_VAR
   VAR CONSTANT
      DB : Byte := 16#84;
   END_VAR
   VAR_TEMP   // added for the SCL form of the ladder/FBD networks
      _w1 : Bool;
      _w2 : Bool;
   END_VAR
BEGIN

REGION Network 1: Initialize Temp Values
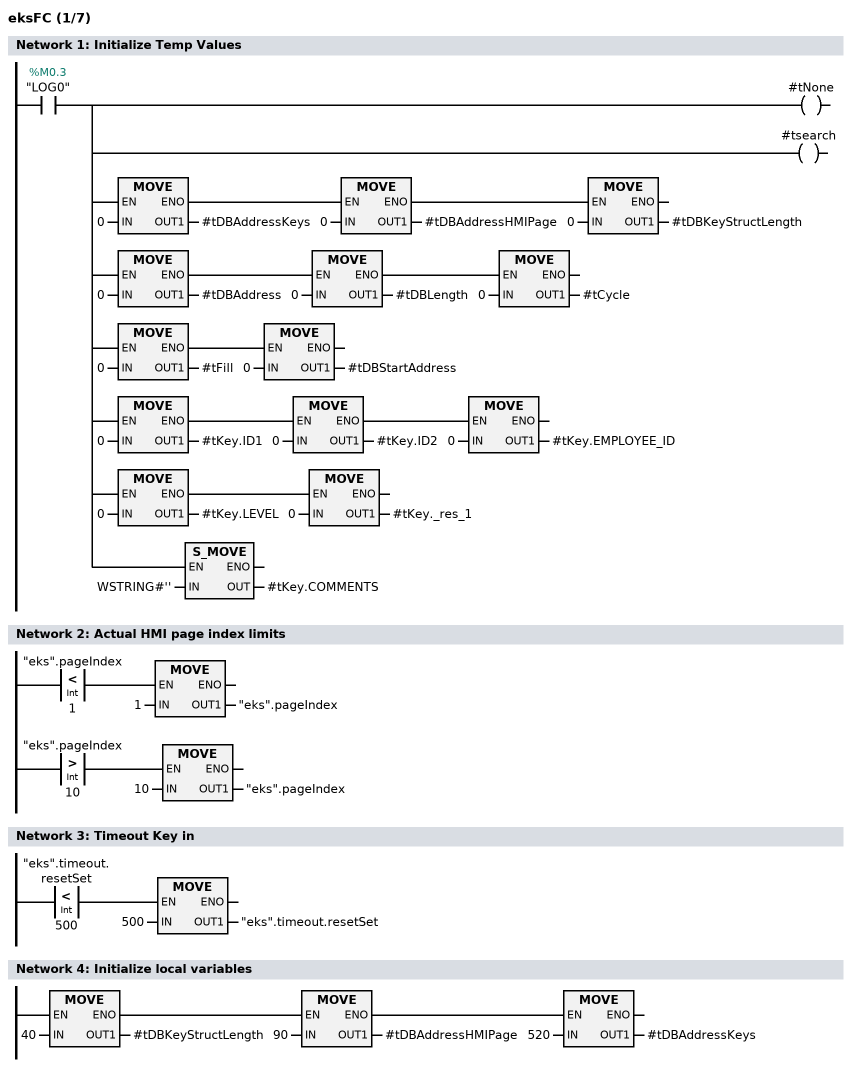
   RUNG wire#powerrail
      Contact( "LOG0" )
      wire#w1
      Coil( #tNone )
   END_RUNG
   RUNG wire#w1
      Coil( #tsearch )
   END_RUNG
   RUNG wire#w1
      Move(in := 0, out1 => #tDBAddressKeys)
      Move(in := 0, out1 => #tDBAddressHMIPage)
      Move(in := 0, out1 => #tDBKeyStructLength)
   END_RUNG
   RUNG wire#w1
      Move(in := 0, out1 => #tDBAddress)
      Move(in := 0, out1 => #tDBLength)
      Move(in := 0, out1 => #tCycle)
   END_RUNG
   RUNG wire#w1
      Move(in := 0, out1 => #tFill)
      Move(in := 0, out1 => #tDBStartAddress)
   END_RUNG
   RUNG wire#w1
      Move(in := 0, out1 => #tKey.ID1)
      Move(in := 0, out1 => #tKey.ID2)
      Move(in := 0, out1 => #tKey.EMPLOYEE_ID)
   END_RUNG
   RUNG wire#w1
      Move(in := 0, out1 => #tKey.LEVEL)
      Move(in := 0, out1 => #tKey._res_1)
   END_RUNG
   RUNG wire#w1
      S_Move(in := WSTRING#'', out => #tKey.COMMENTS)
   END_RUNG
   // the same network as SCL:
   #tNone := "LOG0";
   #tsearch := "LOG0";
   IF "LOG0" THEN
       #tDBAddressKeys := 0;
       #tDBAddressHMIPage := 0;
       #tDBKeyStructLength := 0;
       #tDBAddress := 0;
       #tDBLength := 0;
       #tCycle := 0;
       #tFill := 0;
       #tDBStartAddress := 0;
       #tKey.ID1 := 0;
       #tKey.ID2 := 0;
       #tKey.EMPLOYEE_ID := 0;
       #tKey.LEVEL := 0;
       #tKey._res_1 := 0;
       #tKey.COMMENTS := WSTRING#'';
   END_IF;
END_REGION

REGION Network 2: Actual HMI page index limits
   RUNG wire#powerrail
      { S7_Templates := "SrcType := Int" } LT_Contact(in1 := "eks".pageIndex, in2 := 1)
      Move(in := 1, out1 => "eks".pageIndex)
   END_RUNG
   RUNG wire#powerrail
      { S7_Templates := "SrcType := Int" } GT_Contact(in1 := "eks".pageIndex, in2 := 10)
      Move(in := 10, out1 => "eks".pageIndex)
   END_RUNG
   // the same network as SCL:
   IF "eks".pageIndex < 1 THEN "eks".pageIndex := 1; END_IF;
   IF "eks".pageIndex > 10 THEN "eks".pageIndex := 10; END_IF;
END_REGION

REGION Network 3: Timeout Key in
   RUNG wire#powerrail
      { S7_Templates := "SrcType := Int" } LT_Contact(in1 := "eks".timeout.resetSet, in2 := 500)
      Move(in := 500, out1 => "eks".timeout.resetSet)
   END_RUNG
   // the same network as SCL:
   IF "eks".timeout.resetSet < 500 THEN "eks".timeout.resetSet := 500; END_IF;
END_REGION

REGION Network 4: Initialize local variables
   RUNG wire#powerrail
      Move(in := 40, out1 => #tDBKeyStructLength)
      Move(in := 90, out1 => #tDBAddressHMIPage)
      Move(in := 520, out1 => #tDBAddressKeys)
   END_RUNG
   // the same network as SCL:
   #tDBKeyStructLength := 40;
   #tDBAddressHMIPage := 90;
   #tDBAddressKeys := 520;
END_REGION

REGION Network 6: Calculate data position and length for HMI page
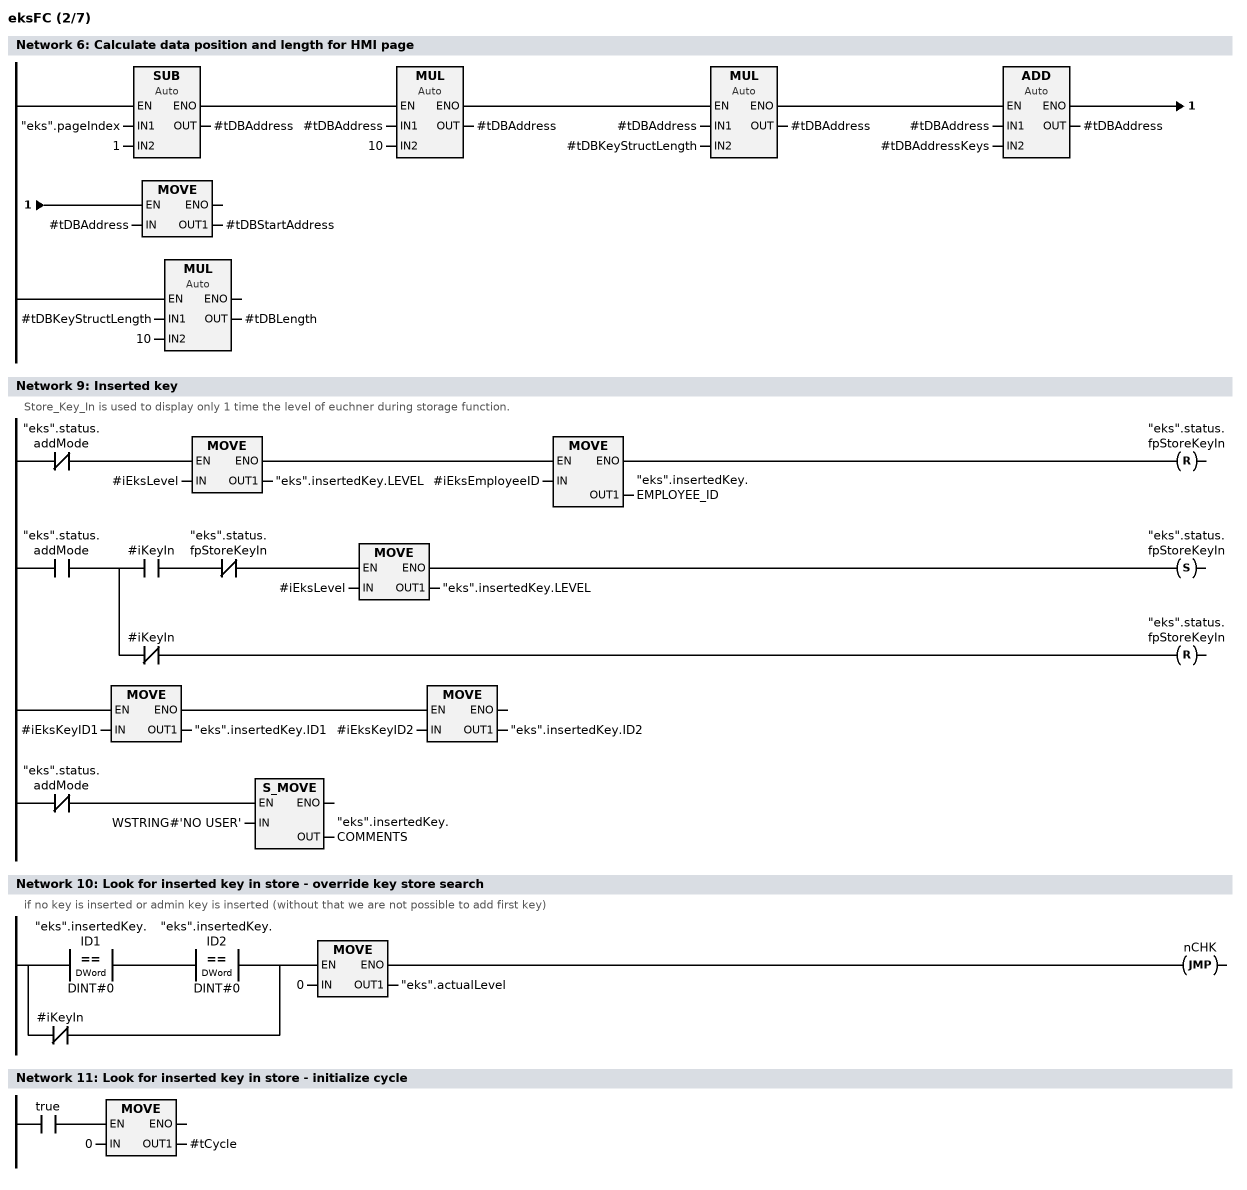
   RUNG wire#powerrail
      Sub(in1 := "eks".pageIndex, in2 := 1, out => #tDBAddress)
      Mul(in1 := #tDBAddress, in2 := 10, out => #tDBAddress)
      Mul(in1 := #tDBAddress, in2 := #tDBKeyStructLength, out => #tDBAddress)
      Add(in1 := #tDBAddress, in2 := #tDBAddressKeys, out => #tDBAddress)
      Move(in := #tDBAddress, out1 => #tDBStartAddress)
   END_RUNG
   RUNG wire#powerrail
      Mul(in1 := #tDBKeyStructLength, in2 := 10, out => #tDBLength)
   END_RUNG
   // the same network as SCL:
   #tDBAddress := "eks".pageIndex - 1;
   #tDBAddress := #tDBAddress * 10;
   #tDBAddress := #tDBAddress * #tDBKeyStructLength;
   #tDBAddress := #tDBAddress + #tDBAddressKeys;
   #tDBStartAddress := #tDBAddress;
   #tDBLength := #tDBKeyStructLength * 10;
END_REGION

REGION Network 7 (SCL): Copy data for page (10 keys)
   POKE_BLK(area_src:=#DB,
            dbNumber_src:=305,
            byteOffset_src:=#tDBAddress,
            area_dest:=#DB,
            dbNumber_dest:=305,
            byteOffset_dest:=90,
            count:=#tDBLength);
END_REGION

REGION Network 9: Inserted key
   // Store_Key_In is used to display only 1 time the level of euchner during storage function.
   RUNG wire#powerrail
      I_Contact( "eks".status.addMode )
      Move(in := #iEksLevel, out1 => "eks".insertedKey.LEVEL)
      Move(in := #iEksEmployeeID, out1 => "eks".insertedKey.EMPLOYEE_ID)
      R_Coil( "eks".status.fpStoreKeyIn )
   END_RUNG
   RUNG wire#powerrail
      Contact( "eks".status.addMode )
      wire#w1
      Contact( #iKeyIn )
      I_Contact( "eks".status.fpStoreKeyIn )
      Move(in := #iEksLevel, out1 => "eks".insertedKey.LEVEL)
      S_Coil( "eks".status.fpStoreKeyIn )
   END_RUNG
   RUNG wire#w1
      I_Contact( #iKeyIn )
      R_Coil( "eks".status.fpStoreKeyIn )
   END_RUNG
   RUNG wire#powerrail
      Move(in := #iEksKeyID1, out1 => "eks".insertedKey.ID1)
      Move(in := #iEksKeyID2, out1 => "eks".insertedKey.ID2)
   END_RUNG
   RUNG wire#powerrail
      I_Contact( "eks".status.addMode )
      S_Move(in := WSTRING#'NO USER', out => "eks".insertedKey.COMMENTS)
   END_RUNG
   // the same network as SCL:
   IF NOT "eks".status.addMode THEN
       "eks".insertedKey.LEVEL := #iEksLevel;
       "eks".insertedKey.EMPLOYEE_ID := #iEksEmployeeID;
       "eks".status.fpStoreKeyIn := FALSE;
   END_IF;
   IF "eks".status.addMode AND #iKeyIn AND NOT "eks".status.fpStoreKeyIn THEN
       "eks".insertedKey.LEVEL := #iEksLevel;
       "eks".status.fpStoreKeyIn := TRUE;
   END_IF;
   IF "eks".status.addMode AND NOT #iKeyIn THEN "eks".status.fpStoreKeyIn := FALSE; END_IF;
   "eks".insertedKey.ID1 := #iEksKeyID1;
   "eks".insertedKey.ID2 := #iEksKeyID2;
   IF NOT "eks".status.addMode THEN "eks".insertedKey.COMMENTS := WSTRING#'NO USER'; END_IF;
END_REGION

REGION Network 10: Look for inserted key in store - override key store search
   // if no key is inserted or admin key is inserted (without that we are not possible to add first key)
   RUNG wire#powerrail
      { S7_Templates := "SrcType := DWord" } EQ_Contact(in1 := "eks".insertedKey.ID1, in2 := DINT#0)
      { S7_Templates := "SrcType := DWord" } EQ_Contact(in1 := "eks".insertedKey.ID2, in2 := DINT#0)
      wire#w1
      Move(in := 0, out1 => "eks".actualLevel)
      JumpCoil( nCHK )
   END_RUNG
   RUNG wire#powerrail
      I_Contact( #iKeyIn )
   END_RUNG wire#w1
   // the same network as SCL:
   #_w1 := (("eks".insertedKey.ID1 = DINT#0) AND ("eks".insertedKey.ID2 = DINT#0)) OR NOT #iKeyIn;
   IF #_w1 THEN
       "eks".actualLevel := 0;
       GOTO nCHK;
   END_IF;
END_REGION

REGION Network 11: Look for inserted key in store - initialize cycle
   RUNG wire#powerrail
      Contact( true )
      Move(in := 0, out1 => #tCycle)
   END_RUNG
   // the same network as SCL:
   IF true THEN #tCycle := 0; END_IF;
END_REGION

REGION Network 12: Look for inserted key in store - calculate data position for key
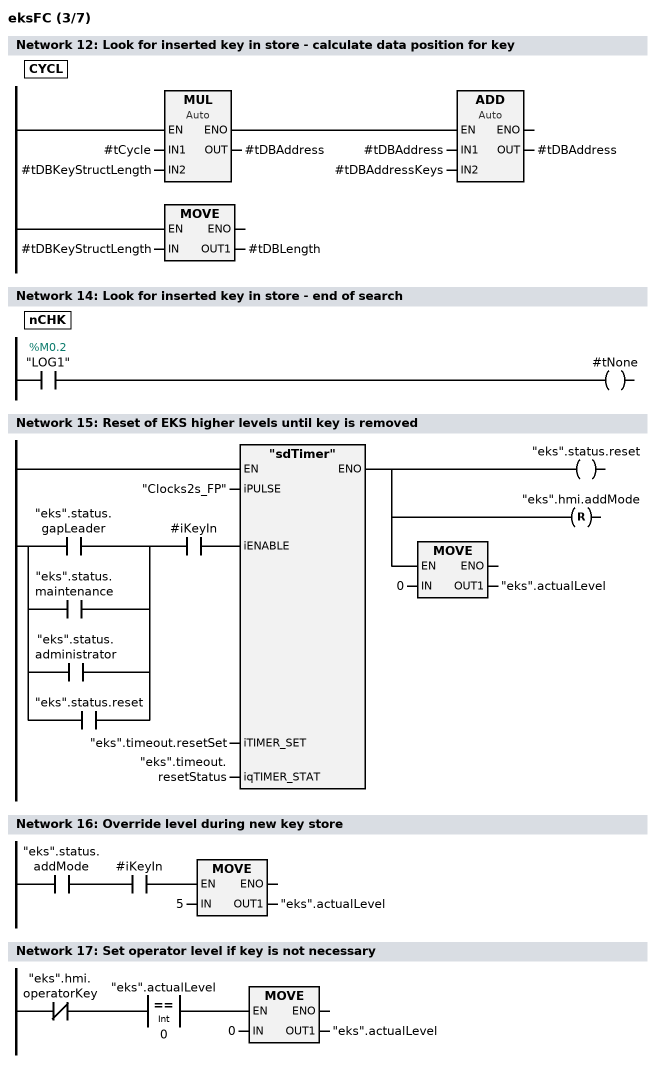
   Label( CYCL )
   RUNG wire#powerrail
      Mul(in1 := #tCycle, in2 := #tDBKeyStructLength, out => #tDBAddress)
      Add(in1 := #tDBAddress, in2 := #tDBAddressKeys, out => #tDBAddress)
   END_RUNG
   RUNG wire#powerrail
      Move(in := #tDBKeyStructLength, out1 => #tDBLength)
   END_RUNG
   // the same network as SCL:
   CYCL:
   #tDBAddress := #tCycle * #tDBKeyStructLength;
   #tDBAddress := #tDBAddress + #tDBAddressKeys;
   #tDBLength := #tDBKeyStructLength;
END_REGION

REGION Network 13 (SCL): Look for inserted key in store - check ID of stored key
   FOR #i := 1 TO 130 DO
       #tKey := "eks".keys[#i];
       IF (#tKey.ID1 = "eks".insertedKey.ID1) AND
           (#tKey.ID2 = "eks".insertedKey.ID2) THEN
           "eks".actualLevel := #tKey.LEVEL;
           "eks".insertedKey.COMMENTS := #tKey.COMMENTS;
           EXIT;
       END_IF;
   END_FOR;
END_REGION

REGION Network 14: Look for inserted key in store - end of search
   Label( nCHK )
   RUNG wire#powerrail
      Contact( "LOG1" )
      Coil( #tNone )
   END_RUNG
   // the same network as SCL:
   nCHK:
   #tNone := "LOG1";
END_REGION

REGION Network 15: Reset of EKS higher levels until key is removed
   RUNG wire#powerrail
      "sdTimer"(iENABLE := wire#w2, iPULSE := "Clocks2s_FP", iTIMER_SET := "eks".timeout.resetSet, iqTIMER_STAT := "eks".timeout.resetStatus)
      wire#w3
      Coil( "eks".status.reset )
   END_RUNG
   RUNG wire#powerrail
      Contact( "eks".status.gapLeader )
      wire#w1
      Contact( #iKeyIn )
   END_RUNG wire#w2
   RUNG wire#powerrail
      Contact( "eks".status.maintenance )
   END_RUNG wire#w1
   RUNG wire#powerrail
      Contact( "eks".status.administrator )
   END_RUNG wire#w1
   RUNG wire#powerrail
      Contact( "eks".status.reset )
   END_RUNG wire#w1
   RUNG wire#w3
      R_Coil( "eks".hmi.addMode )
   END_RUNG
   RUNG wire#w3
      Move(in := 0, out1 => "eks".actualLevel)
   END_RUNG
   // the same network as SCL:
   "sdTimer"(iPULSE := "Clocks2s_FP",
             iENABLE := ("eks".status.gapLeader OR "eks".status.maintenance OR "eks".status.administrator OR "eks".status.reset) AND #iKeyIn,
             iTIMER_SET := "eks".timeout.resetSet,
             iqTIMER_STAT := "eks".timeout.resetStatus,
             ENO => #_w1);
   "eks".status.reset := #_w1;
   IF #_w1 THEN
       "eks".hmi.addMode := FALSE;
       "eks".actualLevel := 0;
   END_IF;
END_REGION

REGION Network 16: Override level during new key store
   RUNG wire#powerrail
      Contact( "eks".status.addMode )
      Contact( #iKeyIn )
      Move(in := 5, out1 => "eks".actualLevel)
   END_RUNG
   // the same network as SCL:
   IF "eks".status.addMode AND #iKeyIn THEN "eks".actualLevel := 5; END_IF;
END_REGION

REGION Network 17: Set operator level if key is not necessary
   RUNG wire#powerrail
      I_Contact( "eks".hmi.operatorKey )
      { S7_Templates := "SrcType := Int" } EQ_Contact(in1 := "eks".actualLevel, in2 := 0)
      Move(in := 0, out1 => "eks".actualLevel)
   END_RUNG
   // the same network as SCL:
   IF NOT "eks".hmi.operatorKey AND ("eks".actualLevel = 0) THEN "eks".actualLevel := 0; END_IF;
END_REGION

REGION Network 18: EKS levels
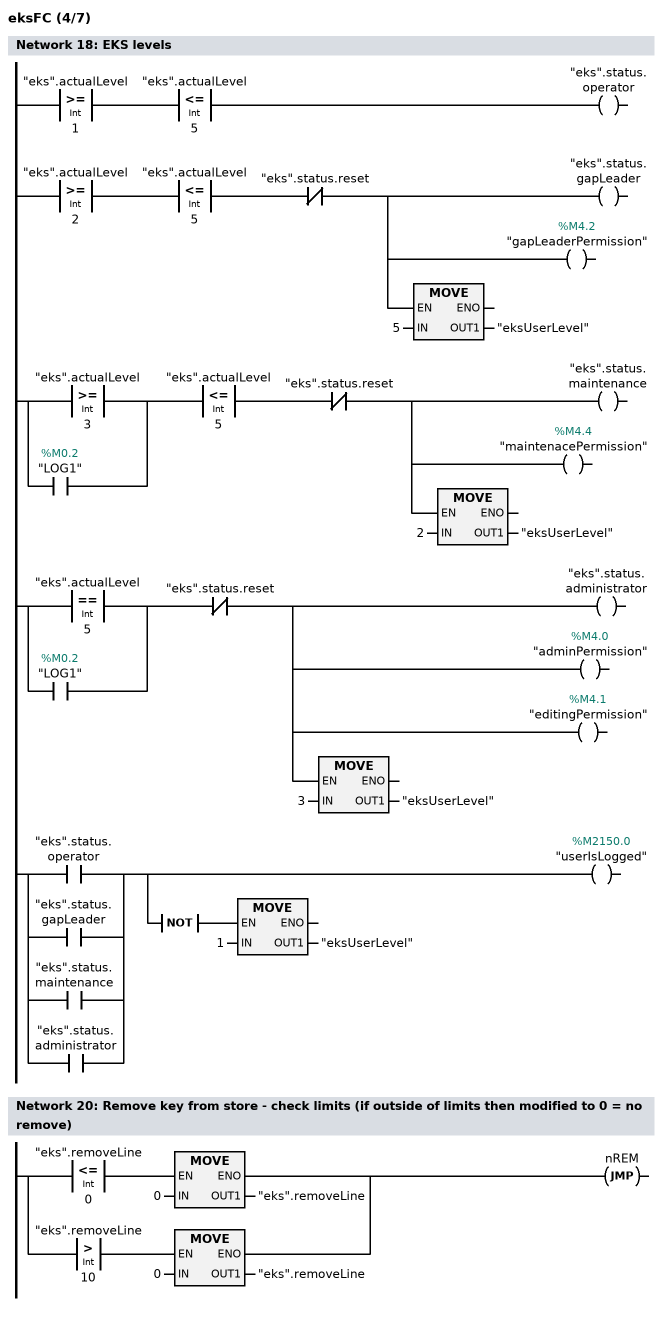
   RUNG wire#powerrail
      { S7_Templates := "SrcType := Int" } GE_Contact(in1 := "eks".actualLevel, in2 := 1)
      { S7_Templates := "SrcType := Int" } LE_Contact(in1 := "eks".actualLevel, in2 := 5)
      Coil( "eks".status.operator )
   END_RUNG
   RUNG wire#powerrail
      { S7_Templates := "SrcType := Int" } GE_Contact(in1 := "eks".actualLevel, in2 := 2)
      { S7_Templates := "SrcType := Int" } LE_Contact(in1 := "eks".actualLevel, in2 := 5)
      I_Contact( "eks".status.reset )
      wire#w1
      Coil( "eks".status.gapLeader )
   END_RUNG
   RUNG wire#w1
      Coil( "gapLeaderPermission" )
   END_RUNG
   RUNG wire#w1
      Move(in := 5, out1 => "eksUserLevel")
   END_RUNG
   RUNG wire#powerrail
      { S7_Templates := "SrcType := Int" } GE_Contact(in1 := "eks".actualLevel, in2 := 3)
      wire#w2
      { S7_Templates := "SrcType := Int" } LE_Contact(in1 := "eks".actualLevel, in2 := 5)
      I_Contact( "eks".status.reset )
      wire#w3
      Coil( "eks".status.maintenance )
   END_RUNG
   RUNG wire#powerrail
      Contact( "LOG1" )
   END_RUNG wire#w2
   RUNG wire#w3
      Coil( "maintenacePermission" )
   END_RUNG
   RUNG wire#w3
      Move(in := 2, out1 => "eksUserLevel")
   END_RUNG
   RUNG wire#powerrail
      { S7_Templates := "SrcType := Int" } EQ_Contact(in1 := "eks".actualLevel, in2 := 5)
      wire#w4
      I_Contact( "eks".status.reset )
      wire#w5
      Coil( "eks".status.administrator )
   END_RUNG
   RUNG wire#powerrail
      Contact( "LOG1" )
   END_RUNG wire#w4
   RUNG wire#w5
      Coil( "adminPermission" )
   END_RUNG
   RUNG wire#w5
      Coil( "editingPermission" )
   END_RUNG
   RUNG wire#w5
      Move(in := 3, out1 => "eksUserLevel")
   END_RUNG
   RUNG wire#powerrail
      Contact( "eks".status.operator )
      wire#w6
      Coil( "userIsLogged" )
   END_RUNG
   RUNG wire#powerrail
      Contact( "eks".status.gapLeader )
   END_RUNG wire#w6
   RUNG wire#powerrail
      Contact( "eks".status.maintenance )
   END_RUNG wire#w6
   RUNG wire#powerrail
      Contact( "eks".status.administrator )
   END_RUNG wire#w6
   RUNG wire#w6
      Not()
      Move(in := 1, out1 => "eksUserLevel")
   END_RUNG
   // the same network as SCL:
   "eks".status.operator := ("eks".actualLevel >= 1) AND ("eks".actualLevel <= 5);
   "eks".status.gapLeader := ("eks".actualLevel >= 2) AND ("eks".actualLevel <= 5) AND NOT "eks".status.reset;
   "gapLeaderPermission" := "eks".status.gapLeader;
   IF "eks".status.gapLeader THEN "eksUserLevel" := 5; END_IF;
   "eks".status.maintenance := (("eks".actualLevel >= 3) OR "LOG1") AND ("eks".actualLevel <= 5) AND NOT "eks".status.reset;
   "maintenacePermission" := "eks".status.maintenance;
   IF "eks".status.maintenance THEN "eksUserLevel" := 2; END_IF;
   "eks".status.administrator := (("eks".actualLevel = 5) OR "LOG1") AND NOT "eks".status.reset;
   "adminPermission" := "eks".status.administrator;
   "editingPermission" := "eks".status.administrator;
   IF "eks".status.administrator THEN "eksUserLevel" := 3; END_IF;
   "userIsLogged" := "eks".status.operator OR "eks".status.gapLeader OR "eks".status.maintenance OR "eks".status.administrator;
   IF NOT "userIsLogged" THEN "eksUserLevel" := 1; END_IF;
END_REGION

REGION Network 20: Remove key from store - check limits (if outside of limits then modified to 0 = no remove)
   RUNG wire#powerrail
      { S7_Templates := "SrcType := Int" } LE_Contact(in1 := "eks".removeLine, in2 := 0)
      Move(in := 0, out1 => "eks".removeLine)
      wire#w1
      JumpCoil( nREM )
   END_RUNG
   RUNG wire#powerrail
      { S7_Templates := "SrcType := Int" } GT_Contact(in1 := "eks".removeLine, in2 := 10)
      Move(in := 0, out1 => "eks".removeLine)
   END_RUNG wire#w1
   // the same network as SCL:
   #_w1 := "eks".removeLine <= 0;
   IF #_w1 THEN "eks".removeLine := 0; END_IF;
   #_w2 := "eks".removeLine > 10;
   IF #_w2 THEN "eks".removeLine := 0; END_IF;
   IF #_w1 OR #_w2 THEN GOTO nREM; END_IF;
END_REGION

REGION Network 21: Remove key from store - calculate data position and length for HMI page
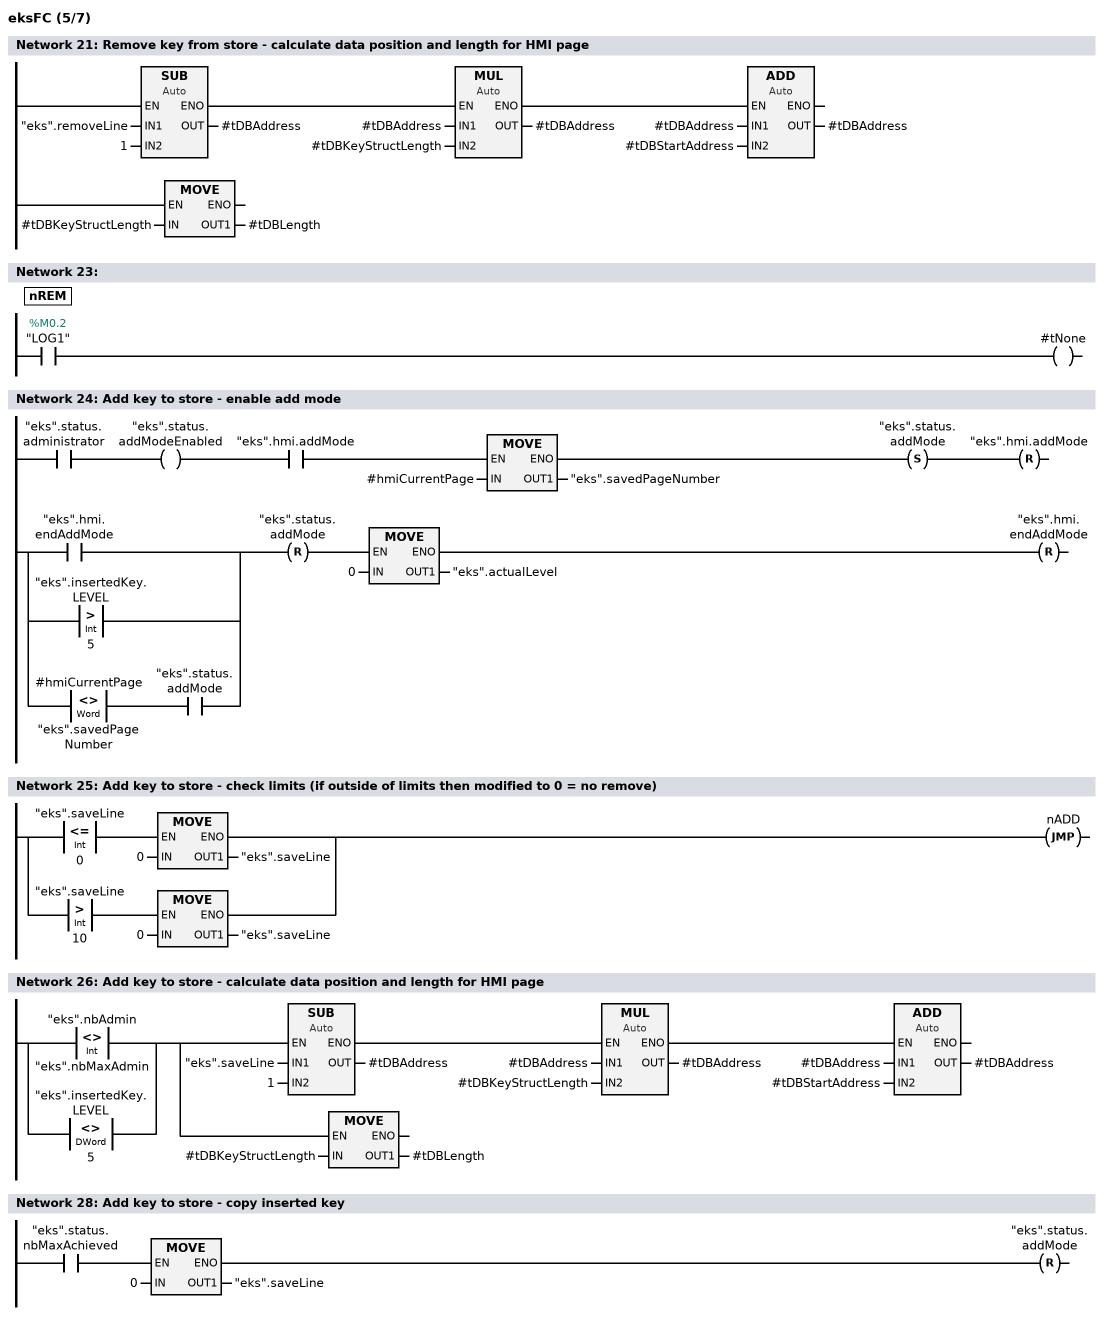
   RUNG wire#powerrail
      Sub(in1 := "eks".removeLine, in2 := 1, out => #tDBAddress)
      Mul(in1 := #tDBAddress, in2 := #tDBKeyStructLength, out => #tDBAddress)
      Add(in1 := #tDBAddress, in2 := #tDBStartAddress, out => #tDBAddress)
   END_RUNG
   RUNG wire#powerrail
      Move(in := #tDBKeyStructLength, out1 => #tDBLength)
   END_RUNG
   // the same network as SCL:
   #tDBAddress := "eks".removeLine - 1;
   #tDBAddress := #tDBAddress * #tDBKeyStructLength;
   #tDBAddress := #tDBAddress + #tDBStartAddress;
   #tDBLength := #tDBKeyStructLength;
END_REGION

REGION Network 22 (SCL): Remove key from store - delete key
   #tFill := 0;

   POKE_BLK(area_src:=#DB,
            dbNumber_src:=305,
            byteOffset_src:=5720,
            area_dest:=#DB,
            dbNumber_dest:=305,
            byteOffset_dest:=#tDBAddress,
            count:=#tDBLength);

   "eks".removeLine := 0;
END_REGION

REGION Network 23
   Label( nREM )
   RUNG wire#powerrail
      Contact( "LOG1" )
      Coil( #tNone )
   END_RUNG
   // the same network as SCL:
   nREM:
   #tNone := "LOG1";
END_REGION

REGION Network 24: Add key to store - enable add mode
   RUNG wire#powerrail
      Contact( "eks".status.administrator )
      Coil( "eks".status.addModeEnabled )
      Contact( "eks".hmi.addMode )
      Move(in := #hmiCurrentPage, out1 => "eks".savedPageNumber)
      S_Coil( "eks".status.addMode )
      R_Coil( "eks".hmi.addMode )
   END_RUNG
   RUNG wire#powerrail
      Contact( "eks".hmi.endAddMode )
      wire#w1
      R_Coil( "eks".status.addMode )
      Move(in := 0, out1 => "eks".actualLevel)
      R_Coil( "eks".hmi.endAddMode )
   END_RUNG
   RUNG wire#powerrail
      { S7_Templates := "SrcType := Int" } GT_Contact(in1 := "eks".insertedKey.LEVEL, in2 := 5)
   END_RUNG wire#w1
   RUNG wire#powerrail
      { S7_Templates := "SrcType := Word" } NE_Contact(in1 := #hmiCurrentPage, in2 := "eks".savedPageNumber)
      Contact( "eks".status.addMode )
   END_RUNG wire#w1
   // the same network as SCL:
   "eks".status.addModeEnabled := "eks".status.administrator;
   IF "eks".status.administrator AND "eks".hmi.addMode THEN
       "eks".savedPageNumber := #hmiCurrentPage;
       "eks".status.addMode := TRUE;
       "eks".hmi.addMode := FALSE;
   END_IF;
   #_w1 := "eks".hmi.endAddMode OR ("eks".insertedKey.LEVEL > 5) OR ((#hmiCurrentPage <> "eks".savedPageNumber) AND "eks".status.addMode);
   IF #_w1 THEN
       "eks".status.addMode := FALSE;
       "eks".actualLevel := 0;
       "eks".hmi.endAddMode := FALSE;
   END_IF;
END_REGION

REGION Network 25: Add key to store - check limits (if outside of limits then modified to 0 = no remove)
   RUNG wire#powerrail
      { S7_Templates := "SrcType := Int" } LE_Contact(in1 := "eks".saveLine, in2 := 0)
      Move(in := 0, out1 => "eks".saveLine)
      wire#w1
      JumpCoil( nADD )
   END_RUNG
   RUNG wire#powerrail
      { S7_Templates := "SrcType := Int" } GT_Contact(in1 := "eks".saveLine, in2 := 10)
      Move(in := 0, out1 => "eks".saveLine)
   END_RUNG wire#w1
   // the same network as SCL:
   #_w1 := "eks".saveLine <= 0;
   IF #_w1 THEN "eks".saveLine := 0; END_IF;
   #_w2 := "eks".saveLine > 10;
   IF #_w2 THEN "eks".saveLine := 0; END_IF;
   IF #_w1 OR #_w2 THEN GOTO nADD; END_IF;
END_REGION

REGION Network 26: Add key to store - calculate data position and length for HMI page
   RUNG wire#powerrail
      { S7_Templates := "SrcType := Int" } NE_Contact(in1 := "eks".nbAdmin, in2 := "eks".nbMaxAdmin)
      wire#w1
      Sub(in1 := "eks".saveLine, in2 := 1, out => #tDBAddress)
      Mul(in1 := #tDBAddress, in2 := #tDBKeyStructLength, out => #tDBAddress)
      Add(in1 := #tDBAddress, in2 := #tDBStartAddress, out => #tDBAddress)
   END_RUNG
   RUNG wire#powerrail
      { S7_Templates := "SrcType := DWord" } NE_Contact(in1 := "eks".insertedKey.LEVEL, in2 := 5)
   END_RUNG wire#w1
   RUNG wire#w1
      Move(in := #tDBKeyStructLength, out1 => #tDBLength)
   END_RUNG
   // the same network as SCL:
   IF ("eks".nbAdmin <> "eks".nbMaxAdmin) OR ("eks".insertedKey.LEVEL <> 5) THEN
       #tDBAddress := "eks".saveLine - 1;
       #tDBAddress := #tDBAddress * #tDBKeyStructLength;
       #tDBAddress := #tDBAddress + #tDBStartAddress;
       #tDBLength := #tDBKeyStructLength;
   END_IF;
END_REGION

REGION Network 27 (SCL): Add key to store - copy inserted key
   IF ("eks".insertedKey.LEVEL = 5  & NOT "eks".status.nbMaxAchieved) OR
       ("eks".insertedKey.LEVEL <> 5) THEN
       POKE_BLK(area_src := #DB,
                dbNumber_src := 305,
                byteOffset_src := 50,
                area_dest := #DB,
                dbNumber_dest := 305,
                byteOffset_dest := #tDBAddress,
                count := #tDBLength);
      "eks".saveLine := 0;
   END_IF;
END_REGION

REGION Network 28: Add key to store - copy inserted key
   RUNG wire#powerrail
      Contact( "eks".status.nbMaxAchieved )
      Move(in := 0, out1 => "eks".saveLine)
      R_Coil( "eks".status.addMode )
   END_RUNG
   // the same network as SCL:
   IF "eks".status.nbMaxAchieved THEN
       "eks".saveLine := 0;
       "eks".status.addMode := FALSE;
   END_IF;
END_REGION

REGION Network 29
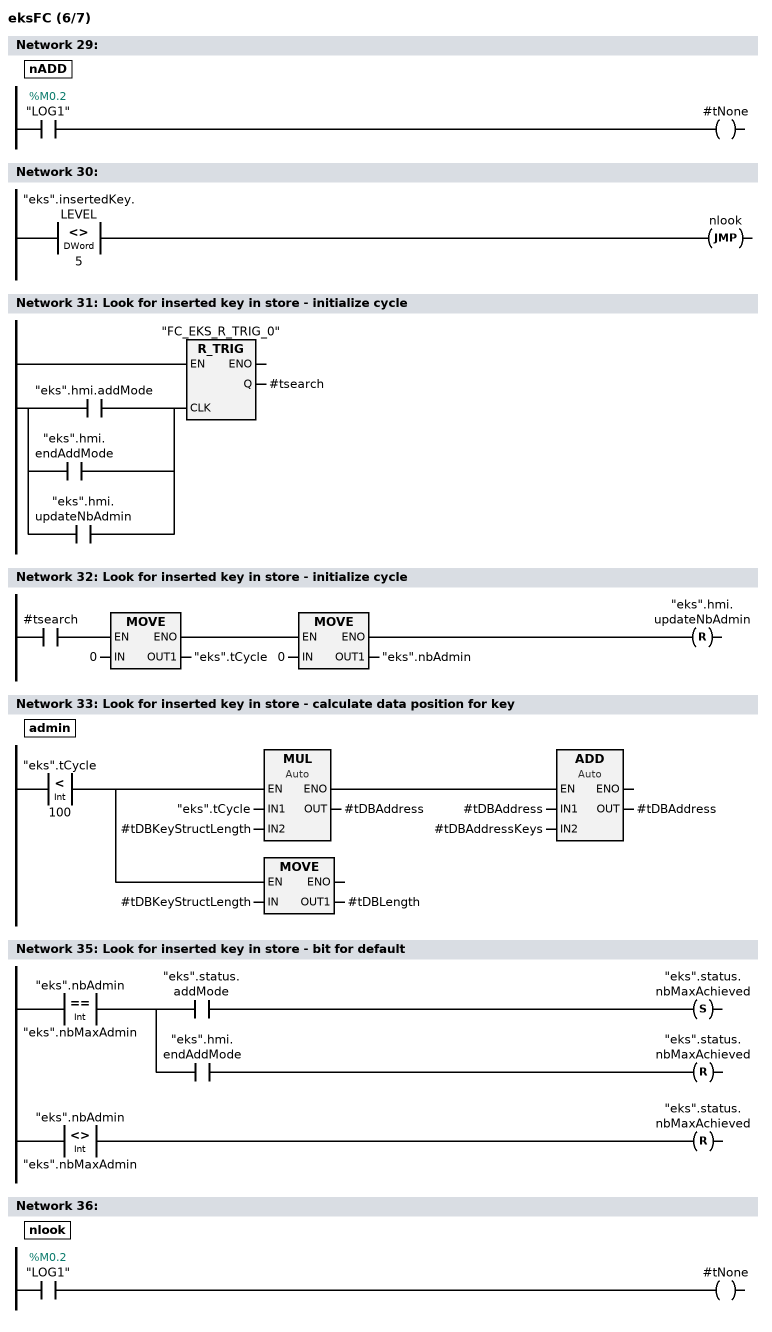
   Label( nADD )
   RUNG wire#powerrail
      Contact( "LOG1" )
      Coil( #tNone )
   END_RUNG
   // the same network as SCL:
   nADD:
   #tNone := "LOG1";
END_REGION

REGION Network 30
   RUNG wire#powerrail
      { S7_Templates := "SrcType := DWord" } NE_Contact(in1 := "eks".insertedKey.LEVEL, in2 := 5)
      JumpCoil( nlook )
   END_RUNG
   // the same network as SCL:
   IF "eks".insertedKey.LEVEL <> 5 THEN GOTO nlook; END_IF;
END_REGION

REGION Network 31: Look for inserted key in store - initialize cycle
   RUNG wire#powerrail
      "FC_EKS_R_TRIG_0".R_TRIG(CLK := wire#w1, Q => #tsearch)
   END_RUNG
   RUNG wire#powerrail
      Contact( "eks".hmi.addMode )
   END_RUNG wire#w1
   RUNG wire#powerrail
      Contact( "eks".hmi.endAddMode )
   END_RUNG wire#w1
   RUNG wire#powerrail
      Contact( "eks".hmi.updateNbAdmin )
   END_RUNG wire#w1
   // the same network as SCL:
   "FC_EKS_R_TRIG_0"(CLK := "eks".hmi.addMode OR "eks".hmi.endAddMode OR "eks".hmi.updateNbAdmin, Q => #tsearch);   // R_TRIG
END_REGION

REGION Network 32: Look for inserted key in store - initialize cycle
   RUNG wire#powerrail
      Contact( #tsearch )
      Move(in := 0, out1 => "eks".tCycle)
      Move(in := 0, out1 => "eks".nbAdmin)
      R_Coil( "eks".hmi.updateNbAdmin )
   END_RUNG
   // the same network as SCL:
   IF #tsearch THEN
       "eks".tCycle := 0;
       "eks".nbAdmin := 0;
       "eks".hmi.updateNbAdmin := FALSE;
   END_IF;
END_REGION

REGION Network 33: Look for inserted key in store - calculate data position for key
   Label( admin )
   RUNG wire#powerrail
      { S7_Templates := "SrcType := Int" } LT_Contact(in1 := "eks".tCycle, in2 := 100)
      wire#w1
      Mul(in1 := "eks".tCycle, in2 := #tDBKeyStructLength, out => #tDBAddress)
      Add(in1 := #tDBAddress, in2 := #tDBAddressKeys, out => #tDBAddress)
   END_RUNG
   RUNG wire#w1
      Move(in := #tDBKeyStructLength, out1 => #tDBLength)
   END_RUNG
   // the same network as SCL:
   admin:
   IF "eks".tCycle < 100 THEN
       #tDBAddress := "eks".tCycle * #tDBKeyStructLength;
       #tDBAddress := #tDBAddress + #tDBAddressKeys;
       #tDBLength := #tDBKeyStructLength;
   END_IF;
END_REGION

REGION Network 34 (SCL): Look for inserted key in store - check ID of stored key
   FOR #i := 1 TO 100 DO
       #tKey := "eks".keys[#i];
       IF #tKey.LEVEL = 5 THEN
           "eks".nbAdmin += 1;
           CONTINUE;
       END_IF;
   END_FOR;
END_REGION

REGION Network 35: Look for inserted key in store - bit for default
   RUNG wire#powerrail
      { S7_Templates := "SrcType := Int" } EQ_Contact(in1 := "eks".nbAdmin, in2 := "eks".nbMaxAdmin)
      wire#w1
      Contact( "eks".status.addMode )
      S_Coil( "eks".status.nbMaxAchieved )
   END_RUNG
   RUNG wire#w1
      Contact( "eks".hmi.endAddMode )
      R_Coil( "eks".status.nbMaxAchieved )
   END_RUNG
   RUNG wire#powerrail
      { S7_Templates := "SrcType := Int" } NE_Contact(in1 := "eks".nbAdmin, in2 := "eks".nbMaxAdmin)
      R_Coil( "eks".status.nbMaxAchieved )
   END_RUNG
   // the same network as SCL:
   #_w1 := "eks".nbAdmin = "eks".nbMaxAdmin;
   IF #_w1 AND "eks".status.addMode THEN "eks".status.nbMaxAchieved := TRUE; END_IF;
   IF #_w1 AND "eks".hmi.endAddMode THEN "eks".status.nbMaxAchieved := FALSE; END_IF;
   IF "eks".nbAdmin <> "eks".nbMaxAdmin THEN "eks".status.nbMaxAchieved := FALSE; END_IF;
END_REGION

REGION Network 36
   Label( nlook )
   RUNG wire#powerrail
      Contact( "LOG1" )
      Coil( #tNone )
   END_RUNG
   // the same network as SCL:
   nlook:
   #tNone := "LOG1";
END_REGION

REGION Network 37: Write Level and Employer ID on Key
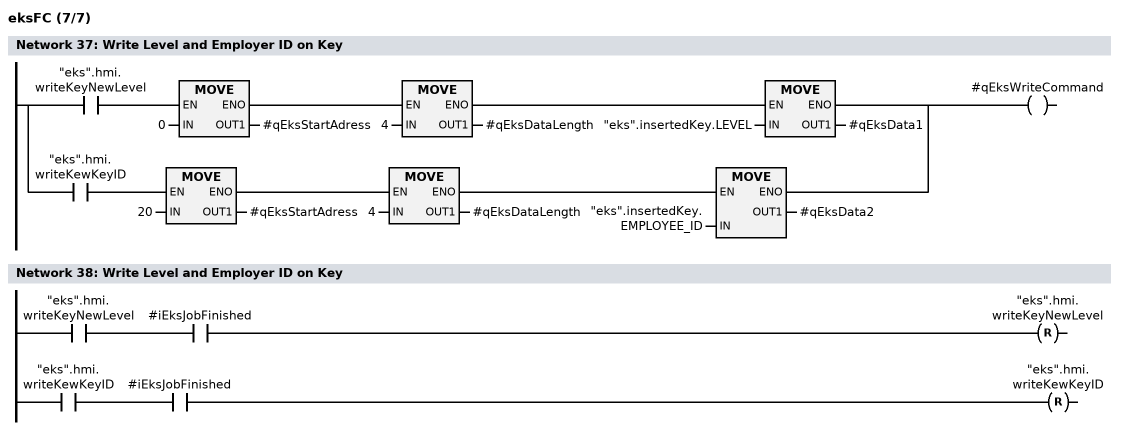
   RUNG wire#powerrail
      Contact( "eks".hmi.writeKeyNewLevel )
      Move(in := 0, out1 => #qEksStartAdress)
      Move(in := 4, out1 => #qEksDataLength)
      Move(in := "eks".insertedKey.LEVEL, out1 => #qEksData1)
      wire#w1
      Coil( #qEksWriteCommand )
   END_RUNG
   RUNG wire#powerrail
      Contact( "eks".hmi.writeKewKeyID )
      Move(in := 20, out1 => #qEksStartAdress)
      Move(in := 4, out1 => #qEksDataLength)
      Move(in := "eks".insertedKey.EMPLOYEE_ID, out1 => #qEksData2)
   END_RUNG wire#w1
   // the same network as SCL:
   IF "eks".hmi.writeKeyNewLevel THEN
       #qEksStartAdress := 0;
       #qEksDataLength := 4;
       #qEksData1 := "eks".insertedKey.LEVEL;
   END_IF;
   IF "eks".hmi.writeKewKeyID THEN
       #qEksStartAdress := 20;
       #qEksDataLength := 4;
       #qEksData2 := "eks".insertedKey.EMPLOYEE_ID;
   END_IF;
   #qEksWriteCommand := "eks".hmi.writeKeyNewLevel OR "eks".hmi.writeKewKeyID;
END_REGION

REGION Network 38: Write Level and Employer ID on Key
   RUNG wire#powerrail
      Contact( "eks".hmi.writeKeyNewLevel )
      Contact( #iEksJobFinished )
      R_Coil( "eks".hmi.writeKeyNewLevel )
   END_RUNG
   RUNG wire#powerrail
      Contact( "eks".hmi.writeKewKeyID )
      Contact( #iEksJobFinished )
      R_Coil( "eks".hmi.writeKewKeyID )
   END_RUNG
   // the same network as SCL:
   IF "eks".hmi.writeKeyNewLevel AND #iEksJobFinished THEN "eks".hmi.writeKeyNewLevel := FALSE; END_IF;
   IF "eks".hmi.writeKewKeyID AND #iEksJobFinished THEN "eks".hmi.writeKewKeyID := FALSE; END_IF;
END_REGION
END_FUNCTION

FUNCTION "sdTimer" : Void   // FC401, LAD
TITLE = Standard simple SD timer
{ S7_Optimized_Access := 'FALSE' }
FAMILY : system
VERSION : 1.0
// stored: AutoNumber false, IsIECCheckEnabled false, SetENOAutomatically false, UDAEnableTagReadback false
   VAR_INPUT
      iPULSE : Bool;   // time impulse
      iENABLE : Bool;   // release of timer
      iTIMER_SET : Int;   // preset value
   END_VAR
   VAR_IN_OUT
      iqTIMER_STAT : Int;   // actual value
   END_VAR
   VAR_TEMP
      tOk : Bool;
   END_VAR
BEGIN

REGION Network 1: If not enabled, then reset actual value of timer
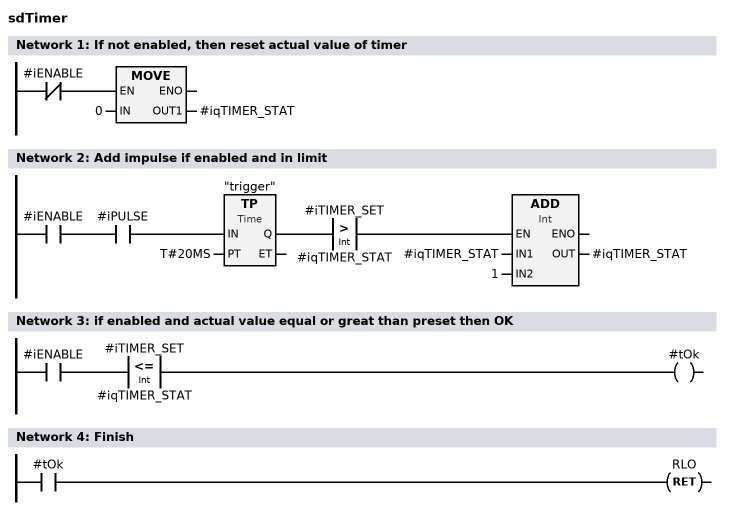
   RUNG wire#powerrail
      I_Contact( #iENABLE )
      { S7_GenerateENO := "TRUE" } Move(in := 0, out1 => #iqTIMER_STAT)
   END_RUNG
   // the same network as SCL:
   IF NOT #iENABLE THEN #iqTIMER_STAT := 0; END_IF;
END_REGION

REGION Network 2: Add impulse if enabled and in limit
   RUNG wire#powerrail
      Contact( #iENABLE )
      Contact( #iPULSE )
      { S7_Templates := "time_type := Time" } "trigger".TP(pt := T#20MS, et =>)
      { S7_Templates := "SrcType := Int" } GT_Contact(in1 := #iTIMER_SET, in2 := #iqTIMER_STAT)
      { S7_Templates := "SrcType := Int"; S7_GenerateENO := "TRUE" } Add(in1 := #iqTIMER_STAT, in2 := 1, out => #iqTIMER_STAT)
   END_RUNG
   // the same network as SCL:
   "trigger".TP(IN := #iENABLE AND #iPULSE, PT := T#20MS);
   IF "trigger".Q AND (#iTIMER_SET > #iqTIMER_STAT) THEN #iqTIMER_STAT := #iqTIMER_STAT + 1; END_IF;
END_REGION

REGION Network 3: if enabled and actual value equal or great than preset then OK
   RUNG wire#powerrail
      Contact( #iENABLE )
      { S7_Templates := "SrcType := Int" } LE_Contact(in1 := #iTIMER_SET, in2 := #iqTIMER_STAT)
      Coil( #tOk )
   END_RUNG
   // the same network as SCL:
   #tOk := #iENABLE AND (#iTIMER_SET <= #iqTIMER_STAT);
END_REGION

REGION Network 4: Finish
   IF #tOk THEN
       ENO := TRUE;
       RETURN;
   END_IF;
END_REGION
END_FUNCTION

FUNCTION "FC_CONTROL_PRINTER" : Void   // FC325, LAD
{ S7_Optimized_Access := 'TRUE' }
VERSION : 0.1
// stored: AutoNumber false, IsIECCheckEnabled false, SetENOAutomatically false, UDAEnableTagReadback false
BEGIN

REGION Network 1
